LIN {X 0.158,Y -379.626,Z 827.651,A 0.000,B 0.000,C 90.000,E1 153.127} C_DIS
LIN {X -0.056,Y -381.140,Z 827.648,A 0.000,B 0.000,C 90.000,E1 152.615} C_DIS
LIN {X 0.104,Y -381.893,Z 827.647,A 0.000,B 0.000,C 90.000,E1 152.410} C_DIS
LIN {X 0.072,Y -384.199,Z 827.643,A 0.000,B 0.000,C 90.000,E1 151.691} C_DIS
LIN {X 0.062,Y -387.788,Z 827.639,A 0.000,B 0.000,C 90.000,E1 150.973} C_DIS
LIN {X 0.027,Y -391.705,Z 827.636,A 0.000,B 0.000,C 90.000,E1 150.383} C_DIS
LIN {X 0.218,Y -394.693,Z 827.634,A 0.000,B 0.000,C 90.000,E1 149.999} C_DIS
LIN {X 0.081,Y -399.557,Z 827.631,A 0.000,B 0.000,C 90.000,E1 149.537} C_DIS
LIN {X -0.054,Y -401.389,Z 827.630,A 0.000,B 0.000,C 90.000,E1 149.410} C_DIS
LIN {X -0.036,Y -407.802,Z 827.628,A 0.000,B 0.000,C 90.000,E1 148.997} C_DIS
LIN {X -0.157,Y -417.907,Z 827.625,A 0.000,B 0.000,C 90.000,E1 148.456} C_DIS
LIN {X -0.139,Y -427.004,Z 827.622,A 0.000,B 0.000,C 90.000,E1 147.995} C_DIS
LIN {X -0.155,Y -435.286,Z 827.620,A 0.000,B 0.000,C 90.000,E1 147.533} C_DIS
LIN {X -0.107,Y -441.668,Z 827.617,A 0.000,B 0.000,C 90.000,E1 147.120} C_DIS
LIN {X 0.193,Y -449.116,Z 827.614,A 0.000,B 0.000,C 90.000,E1 146.501} C_DIS
LIN {X 0.115,Y -453.669,Z 827.612,A 0.000,B 0.000,C 90.000,E1 146.135} C_DIS
LIN {X -0.065,Y -463.952,Z 827.607,A 0.000,B 0.000,C 90.000,E1 145.229} C_DIS
LIN {X -0.066,Y -468.086,Z 827.605,A 0.000,B 0.000,C 90.000,E1 144.815} C_DIS
LIN {X 0.151,Y -473.259,Z 827.601,A 0.000,B 0.000,C 90.000,E1 144.196} C_DIS
LIN {X -0.013,Y -481.998,Z 827.595,A 0.000,B 0.000,C 90.000,E1 143.130} C_DIS
LIN {X 0.058,Y -487.602,Z 827.591,A 0.000,B 0.000,C 90.000,E1 142.351} C_DIS
LIN {X -0.130,Y -494.117,Z 827.586,A 0.000,B 0.000,C 90.000,E1 141.457} C_DIS
LIN {X 0.236,Y -501.224,Z 827.580,A 0.000,B 0.000,C 90.000,E1 140.356} C_DIS
LIN {X 0.094,Y -508.483,Z 827.573,A 0.000,B 0.000,C 90.000,E1 139.175} C_DIS
LIN {X -0.252,Y -513.528,Z 827.568,A 0.000,B 0.000,C 90.000,E1 138.324} C_DIS
LIN {X 0.133,Y -515.933,Z 827.566,A 0.000,B 0.000,C 90.000,E1 137.838} C_DIS
LIN {X 0.247,Y -524.458,Z 827.557,A 0.000,B 0.000,C 90.000,E1 136.215} C_DIS
LIN {X 0.280,Y -528.245,Z 827.553,A 0.000,B 0.000,C 90.000,E1 135.486} C_DIS
LIN {X 0.277,Y -534.712,Z 827.546,A 0.000,B 0.000,C 90.000,E1 134.190} C_DIS
LIN {X 0.004,Y -539.742,Z 827.540,A 0.000,B 0.000,C 90.000,E1 133.218} C_DIS
LIN {X -0.371,Y -546.176,Z 827.532,A 0.000,B 0.000,C 90.000,E1 131.838} C_DIS
LIN {X 0.101,Y -549.719,Z 827.528,A 0.000,B 0.000,C 90.000,E1 130.943} C_DIS
LIN {X -0.174,Y -554.151,Z 827.521,A 0.000,B 0.000,C 90.000,E1 129.850} C_DIS
LIN {X 0.111,Y -558.207,Z 827.515,A 0.000,B 0.000,C 90.000,E1 128.705} C_DIS
LIN {X -0.068,Y -560.940,Z 827.510,A 0.000,B 0.000,C 90.000,E1 127.890} C_DIS
LIN {X -0.225,Y -563.574,Z 827.506,A 0.000,B 0.000,C 90.000,E1 127.076} C_DIS
LIN {X 0.093,Y -565.796,Z 827.501,A 0.000,B 0.000,C 90.000,E1 126.217} C_DIS
LIN {X -0.014,Y -567.045,Z 827.498,A 0.000,B 0.000,C 90.000,E1 125.678} C_DIS
LIN {X -0.327,Y -568.955,Z 827.492,A 0.000,B 0.000,C 90.000,E1 124.612} C_DIS
LIN {X -0.152,Y -570.425,Z 827.486,A 0.000,B 0.000,C 90.000,E1 123.499} C_DIS
LIN {X -0.144,Y -571.632,Z 827.479,A 0.000,B 0.000,C 90.000,E1 122.133} C_DIS
LIN {X -0.372,Y -571.977,Z 827.474,A 0.000,B 0.000,C 90.000,E1 121.337} C_DIS
LIN {X 0.192,Y -571.764,Z 827.469,A 0.000,B 0.000,C 90.000,E1 120.463} C_DIS
LIN {X 0.139,Y -571.928,Z 827.466,A 0.000,B 0.000,C 90.000,E1 119.922} C_DIS
LIN {X -0.198,Y -571.755,Z 827.463,A 0.000,B 0.000,C 90.000,E1 119.411} C_DIS
LIN {X 0.245,Y -571.352,Z 827.460,A 0.000,B 0.000,C 90.000,E1 118.821} C_DIS
LIN {X 0.182,Y -570.016,Z 827.453,A 0.000,B 0.000,C 90.000,E1 117.462} C_DIS
LIN {X 0.013,Y -569.716,Z 827.451,A 0.000,B 0.000,C 90.000,E1 117.206} C_DIS
LIN {X 0.264,Y -568.037,Z 827.447,A 0.000,B 0.000,C 90.000,E1 116.360} C_DIS
LIN {X -0.266,Y -566.017,Z 827.442,A 0.000,B 0.000,C 90.000,E1 115.591} C_DIS
LIN {X 0.063,Y -565.403,Z 827.441,A 0.000,B 0.000,C 90.000,E1 115.283} C_DIS
LIN {X -0.077,Y -562.630,Z 827.435,A 0.000,B 0.000,C 90.000,E1 114.335} C_DIS
LIN {X -0.174,Y -562.501,Z 827.434,A 0.000,B 0.000,C 90.000,E1 114.207} C_DIS
LIN {X 0.056,Y -562.518,Z 827.434,A 0.000,B 0.000,C 90.000,E1 114.027} C_DIS
LIN {X -0.142,Y -562.013,Z 827.432,A 0.000,B 0.000,C 90.000,E1 113.770} C_DIS
LIN {X 0.177,Y -562.133,Z 827.430,A 0.000,B 0.000,C 90.000,E1 113.462} C_DIS
LIN {X -0.023,Y -561.934,Z 827.429,A 0.000,B 0.000,C 90.000,E1 113.206} C_DIS
LIN {X -0.063,Y -561.520,Z 827.428,A 0.000,B 0.000,C 90.000,E1 113.003} C_DIS
LIN {X 0.091,Y -561.775,Z 827.426,A 0.000,B 0.000,C 90.000,E1 112.642} C_DIS
LIN {X -0.213,Y -561.989,Z 827.421,A 0.000,B 0.000,C 90.000,E1 111.844} C_DIS
LIN {X 0.214,Y -562.412,Z 827.417,A 0.000,B 0.000,C 90.000,E1 110.972} C_DIS
LIN {X -0.173,Y -562.591,Z 827.409,A 0.000,B 0.000,C 90.000,E1 109.631} C_DIS
LIN {X -0.201,Y -562.482,Z 827.395,A 0.000,B 0.000,C 90.000,E1 107.149} C_DIS
LIN {X -0.108,Y -563.355,Z 827.377,A 0.000,B 0.000,C 90.000,E1 103.828} C_DIS
LIN {X -0.124,Y -564.958,Z 827.362,A 0.000,B 0.000,C 90.000,E1 101.074} C_DIS
LIN {X -0.229,Y -566.219,Z 827.352,A 0.000,B 0.000,C 90.000,E1 99.434} C_DIS
LIN {X 0.057,Y -567.336,Z 827.343,A 0.000,B 0.000,C 90.000,E1 97.757} C_DIS
LIN {X -0.261,Y -568.305,Z 827.334,A 0.000,B 0.000,C 90.000,E1 96.144} C_DIS
LIN {X -0.106,Y -568.991,Z 827.326,A 0.000,B 0.000,C 90.000,E1 94.759} C_DIS
LIN {X -0.036,Y -569.598,Z 827.319,A 0.000,B 0.000,C 90.000,E1 93.383} C_DIS
LIN {X 0.057,Y -570.037,Z 827.311,A 0.000,B 0.000,C 90.000,E1 92.007} C_DIS
LIN {X 0.154,Y -570.510,Z 827.304,A 0.000,B 0.000,C 90.000,E1 90.630} C_DIS
LIN {X -0.193,Y -570.931,Z 827.295,A 0.000,B 0.000,C 90.000,E1 89.026} C_DIS
LIN {X -0.082,Y -571.308,Z 827.287,A 0.000,B 0.000,C 90.000,E1 87.650} C_DIS
LIN {X -0.236,Y -571.670,Z 827.276,A 0.000,B 0.000,C 90.000,E1 85.755} C_DIS
LIN {X -0.073,Y -571.889,Z 827.269,A 0.000,B 0.000,C 90.000,E1 84.375} C_DIS
LIN {X 0.271,Y -572.275,Z 827.260,A 0.000,B 0.000,C 90.000,E1 82.704} C_DIS
LIN {X -0.052,Y -572.772,Z 827.248,A 0.000,B 0.000,C 90.000,E1 80.557} C_DIS
LIN {X 0.274,Y -573.188,Z 827.240,A 0.000,B 0.000,C 90.000,E1 79.162} C_DIS
LIN {X 0.031,Y -573.590,Z 827.232,A 0.000,B 0.000,C 90.000,E1 77.825} C_DIS
LIN {X 0.038,Y -573.823,Z 827.225,A 0.000,B 0.000,C 90.000,E1 76.464} C_DIS
LIN {X 0.257,Y -574.035,Z 827.216,A 0.000,B 0.000,C 90.000,E1 74.810} C_DIS
LIN {X -0.278,Y -574.043,Z 827.208,A 0.000,B 0.000,C 90.000,E1 73.504} C_DIS
LIN {X -0.103,Y -574.028,Z 827.201,A 0.000,B 0.000,C 90.000,E1 72.127} C_DIS
LIN {X 0.249,Y -573.869,Z 827.193,A 0.000,B 0.000,C 90.000,E1 70.732} C_DIS
LIN {X 0.047,Y -573.554,Z 827.183,A 0.000,B 0.000,C 90.000,E1 68.847} C_DIS
LIN {X -0.112,Y -573.131,Z 827.173,A 0.000,B 0.000,C 90.000,E1 67.230} C_DIS
LIN {X -0.112,Y -572.685,Z 827.166,A 0.000,B 0.000,C 90.000,E1 65.869} C_DIS
LIN {X -0.250,Y -572.259,Z 827.160,A 0.000,B 0.000,C 90.000,E1 64.793} C_DIS
LIN {X 0.044,Y -571.456,Z 827.151,A 0.000,B 0.000,C 90.000,E1 63.127} C_DIS
LIN {X -0.018,Y -570.640,Z 827.143,A 0.000,B 0.000,C 90.000,E1 61.769} C_DIS
LIN {X 0.073,Y -569.770,Z 827.137,A 0.000,B 0.000,C 90.000,E1 60.667} C_DIS
LIN {X -0.171,Y -568.952,Z 827.133,A 0.000,B 0.000,C 90.000,E1 59.871} C_DIS
LIN {X 0.173,Y -567.724,Z 827.126,A 0.000,B 0.000,C 90.000,E1 58.742} C_DIS
LIN {X 0.014,Y -566.317,Z 827.120,A 0.000,B 0.000,C 90.000,E1 57.661} C_DIS
LIN {X 0.144,Y -564.684,Z 827.114,A 0.000,B 0.000,C 90.000,E1 56.548} C_DIS
LIN {X 0.152,Y -563.325,Z 827.110,A 0.000,B 0.000,C 90.000,E1 55.722} C_DIS
LIN {X 0.143,Y -561.776,Z 827.105,A 0.000,B 0.000,C 90.000,E1 54.895} C_DIS
LIN {X 0.206,Y -559.363,Z 827.099,A 0.000,B 0.000,C 90.000,E1 53.783} C_DIS
LIN {X 0.030,Y -557.395,Z 827.094,A 0.000,B 0.000,C 90.000,E1 52.970} C_DIS
LIN {X 0.200,Y -555.953,Z 827.091,A 0.000,B 0.000,C 90.000,E1 52.396} C_DIS
LIN {X -0.002,Y -553.554,Z 827.087,A 0.000,B 0.000,C 90.000,E1 51.582} C_DIS
LIN {X 0.203,Y -550.838,Z 827.082,A 0.000,B 0.000,C 90.000,E1 50.723} C_DIS
LIN {X -0.053,Y -547.802,Z 827.077,A 0.000,B 0.000,C 90.000,E1 49.908} C_DIS
LIN {X 0.035,Y -545.676,Z 827.074,A 0.000,B 0.000,C 90.000,E1 49.337} C_DIS
LIN {X 0.077,Y -541.954,Z 827.069,A 0.000,B 0.000,C 90.000,E1 48.485} C_DIS
LIN {X 0.066,Y -539.294,Z 827.066,A 0.000,B 0.000,C 90.000,E1 47.919} C_DIS
LIN {X -0.320,Y -536.391,Z 827.063,A 0.000,B 0.000,C 90.000,E1 47.391} C_DIS
LIN {X 0.198,Y -532.300,Z 827.059,A 0.000,B 0.000,C 90.000,E1 46.620} C_DIS
LIN {X 0.126,Y -528.699,Z 827.056,A 0.000,B 0.000,C 90.000,E1 46.053} C_DIS
LIN {X 0.029,Y -524.808,Z 827.053,A 0.000,B 0.000,C 90.000,E1 45.486} C_DIS
LIN {X -0.089,Y -520.511,Z 827.050,A 0.000,B 0.000,C 90.000,E1 44.919} C_DIS
LIN {X -0.014,Y -517.102,Z 827.047,A 0.000,B 0.000,C 90.000,E1 44.474} C_DIS
LIN {X 0.175,Y -512.157,Z 827.044,A 0.000,B 0.000,C 90.000,E1 43.866} C_DIS
LIN {X 0.016,Y -506.901,Z 827.041,A 0.000,B 0.000,C 90.000,E1 43.299} C_DIS
LIN {X 0.165,Y -502.891,Z 827.038,A 0.000,B 0.000,C 90.000,E1 42.852} C_DIS
LIN {X -0.018,Y -494.404,Z 827.034,A 0.000,B 0.000,C 90.000,E1 42.043} C_DIS
LIN {X -0.116,Y -486.930,Z 827.030,A 0.000,B 0.000,C 90.000,E1 41.391} C_DIS
LIN {X 0.099,Y -477.756,Z 827.026,A 0.000,B 0.000,C 90.000,E1 40.620} C_DIS
LIN {X 0.063,Y -469.888,Z 827.022,A 0.000,B 0.000,C 90.000,E1 40.011} C_DIS
LIN {X 0.018,Y -458.832,Z 827.018,A 0.000,B 0.000,C 90.000,E1 39.197} C_DIS
LIN {X 0.144,Y -442.903,Z 827.011,A 0.000,B 0.000,C 90.000,E1 38.016} C_DIS
LIN {X -0.087,Y -419.409,Z 827.001,A 0.000,B 0.000,C 90.000,E1 36.217} C_DIS
LIN {X -0.110,Y -405.927,Z 826.995,A 0.000,B 0.000,C 90.000,E1 35.025} C_DIS
LIN {X -0.100,Y -400.639,Z 826.992,A 0.000,B 0.000,C 90.000,E1 34.485} C_DIS
LIN {X 0.175,Y -397.087,Z 826.989,A 0.000,B 0.000,C 90.000,E1 33.992} C_DIS
LIN {X 0.136,Y -397.070,Z 826.989,A 0.000,B 0.000,C 90.000,E1 33.992} C_DIS
LIN {X 0.141,Y -393.525,Z 826.976,A 0.000,B 0.000,C 90.000,E1 31.671} C_DIS
LIN {X 0.136,Y -391.963,Z 826.972,A 0.000,B 0.000,C 90.000,E1 30.875} C_DIS
LIN {X 0.067,Y -391.882,Z 826.971,A 0.000,B 0.000,C 90.000,E1 30.797} C_DIS
LIN {X 0.021,Y -393.684,Z 826.951,A 0.000,B 0.000,C 90.000,E1 27.078} C_DIS
LIN {X -0.061,Y -395.561,Z 826.935,A 0.000,B 0.000,C 90.000,E1 24.259} C_DIS
LIN {X -0.131,Y -397.199,Z 826.923,A 0.000,B 0.000,C 90.000,E1 22.153} C_DIS
LIN {X -0.014,Y -399.623,Z 826.907,A 0.000,B 0.000,C 90.000,E1 19.322} C_DIS
LIN {X 0.166,Y -402.678,Z 826.892,A 0.000,B 0.000,C 90.000,E1 16.496} C_DIS
LIN {X -0.165,Y -407.528,Z 826.872,A 0.000,B 0.000,C 90.000,E1 13.063} C_DIS
LIN {X 0.173,Y -412.017,Z 826.857,A 0.000,B 0.000,C 90.000,E1 10.254} C_DIS
LIN {X -0.001,Y -415.629,Z 826.846,A 0.000,B 0.000,C 90.000,E1 8.219} C_DIS
LIN {X 0.199,Y -418.690,Z 826.836,A 0.000,B 0.000,C 90.000,E1 6.486} C_DIS
LIN {X 0.057,Y -423.009,Z 826.823,A 0.000,B 0.000,C 90.000,E1 4.131} C_DIS
LIN {X 0.036,Y -427.709,Z 826.810,A 0.000,B 0.000,C 90.000,E1 1.776} C_DIS
LIN {X -0.020,Y -434.217,Z 826.793,A 0.000,B 0.000,C 90.000,E1 358.797} C_DIS
LIN {X 0.151,Y -438.864,Z 826.782,A 0.000,B 0.000,C 90.000,E1 356.788} C_DIS
LIN {X -0.116,Y -442.925,Z 826.773,A 0.000,B 0.000,C 90.000,E1 355.179} C_DIS
LIN {X -0.142,Y -447.878,Z 826.762,A 0.000,B 0.000,C 90.000,E1 353.223} C_DIS
LIN {X -0.146,Y -452.367,Z 826.753,A 0.000,B 0.000,C 90.000,E1 351.602} C_DIS
LIN {X 0.126,Y -454.113,Z 826.751,A 0.000,B 0.000,C 90.000,E1 351.084} C_DIS
LIN {X -0.113,Y -455.583,Z 826.749,A 0.000,B 0.000,C 90.000,E1 350.792} C_DIS
LIN {X -0.042,Y -456.513,Z 826.748,A 0.000,B 0.000,C 90.000,E1 350.622} C_DIS
LIN {X 0.095,Y -458.920,Z 826.746,A 0.000,B 0.000,C 90.000,E1 350.274} C_DIS
LIN {X -0.144,Y -461.863,Z 826.744,A 0.000,B 0.000,C 90.000,E1 349.982} C_DIS
LIN {X 0.139,Y -467.280,Z 826.742,A 0.000,B 0.000,C 90.000,E1 349.511} C_DIS
LIN {X -0.155,Y -475.770,Z 826.739,A 0.000,B 0.000,C 90.000,E1 348.993} C_DIS
LIN {X -0.103,Y -488.891,Z 826.734,A 0.000,B 0.000,C 90.000,E1 348.173} C_DIS
LIN {X 0.094,Y -504.918,Z 826.729,A 0.000,B 0.000,C 90.000,E1 347.117} C_DIS
LIN {X -0.200,Y -514.264,Z 826.725,A 0.000,B 0.000,C 90.000,E1 346.520} C_DIS
LIN {X -0.122,Y -526.667,Z 826.720,A 0.000,B 0.000,C 90.000,E1 345.644} C_DIS
LIN {X -0.231,Y -535.675,Z 826.717,A 0.000,B 0.000,C 90.000,E1 344.991} C_DIS
LIN {X -0.012,Y -544.484,Z 826.713,A 0.000,B 0.000,C 90.000,E1 344.283} C_DIS
LIN {X 0.043,Y -551.586,Z 826.709,A 0.000,B 0.000,C 90.000,E1 343.685} C_DIS
LIN {X -0.135,Y -558.409,Z 826.706,A 0.000,B 0.000,C 90.000,E1 343.087} C_DIS
LIN {X 0.238,Y -563.727,Z 826.703,A 0.000,B 0.000,C 90.000,E1 342.543} C_DIS
LIN {X -0.314,Y -570.002,Z 826.700,A 0.000,B 0.000,C 90.000,E1 341.945} C_DIS
LIN {X -0.233,Y -574.905,Z 826.697,A 0.000,B 0.000,C 90.000,E1 341.402} C_DIS
LIN {X 0.043,Y -578.475,Z 826.694,A 0.000,B 0.000,C 90.000,E1 340.967} C_DIS
LIN {X -0.278,Y -584.902,Z 826.690,A 0.000,B 0.000,C 90.000,E1 340.188} C_DIS
LIN {X -0.276,Y -589.853,Z 826.686,A 0.000,B 0.000,C 90.000,E1 339.518} C_DIS
LIN {X -0.018,Y -594.338,Z 826.682,A 0.000,B 0.000,C 90.000,E1 338.827} C_DIS
LIN {X -0.244,Y -600.170,Z 826.677,A 0.000,B 0.000,C 90.000,E1 337.922} C_DIS
LIN {X 0.050,Y -605.603,Z 826.672,A 0.000,B 0.000,C 90.000,E1 336.975} C_DIS
LIN {X 0.157,Y -611.642,Z 826.666,A 0.000,B 0.000,C 90.000,E1 335.921} C_DIS
LIN {X -0.212,Y -616.711,Z 826.661,A 0.000,B 0.000,C 90.000,E1 335.049} C_DIS
LIN {X -0.268,Y -622.133,Z 826.656,A 0.000,B 0.000,C 90.000,E1 334.024} C_DIS
LIN {X -0.258,Y -625.952,Z 826.651,A 0.000,B 0.000,C 90.000,E1 333.256} C_DIS
LIN {X -0.212,Y -629.576,Z 826.647,A 0.000,B 0.000,C 90.000,E1 332.487} C_DIS
LIN {X 0.235,Y -635.207,Z 826.640,A 0.000,B 0.000,C 90.000,E1 331.179} C_DIS
LIN {X -0.192,Y -638.553,Z 826.636,A 0.000,B 0.000,C 90.000,E1 330.461} C_DIS
LIN {X -0.210,Y -642.760,Z 826.630,A 0.000,B 0.000,C 90.000,E1 329.459} C_DIS
LIN {X 0.313,Y -645.746,Z 826.626,A 0.000,B 0.000,C 90.000,E1 328.663} C_DIS
LIN {X -0.157,Y -649.350,Z 826.621,A 0.000,B 0.000,C 90.000,E1 327.709} C_DIS
LIN {X -0.037,Y -652.768,Z 826.615,A 0.000,B 0.000,C 90.000,E1 326.707} C_DIS
LIN {X 0.029,Y -656.724,Z 826.608,A 0.000,B 0.000,C 90.000,E1 325.468} C_DIS
LIN {X 0.040,Y -658.162,Z 826.605,A 0.000,B 0.000,C 90.000,E1 324.975} C_DIS
LIN {X 0.092,Y -660.874,Z 826.600,A 0.000,B 0.000,C 90.000,E1 323.989} C_DIS
LIN {X 0.176,Y -663.377,Z 826.595,A 0.000,B 0.000,C 90.000,E1 323.004} C_DIS
LIN {X -0.267,Y -666.235,Z 826.588,A 0.000,B 0.000,C 90.000,E1 321.823} C_DIS
LIN {X -0.216,Y -667.749,Z 826.584,A 0.000,B 0.000,C 90.000,E1 321.090} C_DIS
LIN {X -0.073,Y -670.596,Z 826.576,A 0.000,B 0.000,C 90.000,E1 319.622} C_DIS
LIN {X 0.031,Y -672.703,Z 826.569,A 0.000,B 0.000,C 90.000,E1 318.405} C_DIS
LIN {X -0.351,Y -674.357,Z 826.564,A 0.000,B 0.000,C 90.000,E1 317.472} C_DIS
LIN {X 0.215,Y -675.447,Z 826.560,A 0.000,B 0.000,C 90.000,E1 316.701} C_DIS
LIN {X 0.366,Y -677.090,Z 826.553,A 0.000,B 0.000,C 90.000,E1 315.486} C_DIS
LIN {X -0.008,Y -678.029,Z 826.549,A 0.000,B 0.000,C 90.000,E1 314.798} C_DIS
LIN {X -0.213,Y -679.943,Z 826.540,A 0.000,B 0.000,C 90.000,E1 313.137} C_DIS
LIN {X 0.084,Y -681.575,Z 826.532,A 0.000,B 0.000,C 90.000,E1 311.676} C_DIS
LIN {X 0.368,Y -682.868,Z 826.525,A 0.000,B 0.000,C 90.000,E1 310.458} C_DIS
LIN {X -0.337,Y -683.813,Z 826.520,A 0.000,B 0.000,C 90.000,E1 309.564} C_DIS
LIN {X 0.118,Y -685.070,Z 826.512,A 0.000,B 0.000,C 90.000,E1 308.096} C_DIS
LIN {X -0.194,Y -686.524,Z 826.503,A 0.000,B 0.000,C 90.000,E1 306.457} C_DIS
LIN {X 0.264,Y -687.475,Z 826.496,A 0.000,B 0.000,C 90.000,E1 305.231} C_DIS
LIN {X -0.055,Y -688.329,Z 826.489,A 0.000,B 0.000,C 90.000,E1 304.072} C_DIS
LIN {X 0.093,Y -689.695,Z 826.479,A 0.000,B 0.000,C 90.000,E1 302.163} C_DIS
LIN {X 0.045,Y -690.732,Z 826.471,A 0.000,B 0.000,C 90.000,E1 300.747} C_DIS
LIN {X 0.001,Y -691.745,Z 826.463,A 0.000,B 0.000,C 90.000,E1 299.333} C_DIS
LIN {X 0.230,Y -692.758,Z 826.455,A 0.000,B 0.000,C 90.000,E1 297.897} C_DIS
LIN {X -0.216,Y -694.091,Z 826.446,A 0.000,B 0.000,C 90.000,E1 296.283} C_DIS
LIN {X 0.106,Y -695.069,Z 826.439,A 0.000,B 0.000,C 90.000,E1 295.079} C_DIS
LIN {X -0.062,Y -695.667,Z 826.435,A 0.000,B 0.000,C 90.000,E1 294.387} C_DIS
LIN {X -0.224,Y -695.703,Z 826.432,A 0.000,B 0.000,C 90.000,E1 293.695} C_DIS
LIN {X 0.001,Y -694.815,Z 826.429,A 0.000,B 0.000,C 90.000,E1 293.206} C_DIS
LIN {X 0.249,Y -694.146,Z 826.428,A 0.000,B 0.000,C 90.000,E1 292.950} C_DIS
LIN {X 0.226,Y -692.688,Z 826.426,A 0.000,B 0.000,C 90.000,E1 292.717} C_DIS
LIN {X -0.055,Y -689.883,Z 826.424,A 0.000,B 0.000,C 90.000,E1 292.386} C_DIS
LIN {X -0.201,Y -688.713,Z 826.424,A 0.000,B 0.000,C 90.000,E1 292.280} C_DIS
LIN {X -0.087,Y -686.910,Z 826.423,A 0.000,B 0.000,C 90.000,E1 292.153} C_DIS
LIN {X 0.187,Y -681.422,Z 826.422,A 0.000,B 0.000,C 90.000,E1 291.844} C_DIS
LIN {X 0.130,Y -679.603,Z 826.421,A 0.000,B 0.000,C 90.000,E1 291.770} C_DIS
LIN {X 0.095,Y -671.476,Z 826.420,A 0.000,B 0.000,C 90.000,E1 291.535} C_DIS
LIN {X -0.183,Y -663.435,Z 826.419,A 0.000,B 0.000,C 90.000,E1 291.408} C_DIS
LIN {X 0.147,Y -650.714,Z 826.418,A 0.000,B 0.000,C 90.000,E1 291.173} C_DIS
LIN {X 0.197,Y -640.689,Z 826.417,A 0.000,B 0.000,C 90.000,E1 290.972} C_DIS
LIN {X -0.266,Y -631.460,Z 826.415,A 0.000,B 0.000,C 90.000,E1 290.791} C_DIS
LIN {X 0.177,Y -628.223,Z 826.415,A 0.000,B 0.000,C 90.000,E1 290.663} C_DIS
LIN {X -0.027,Y -621.652,Z 826.414,A 0.000,B 0.000,C 90.000,E1 290.429} C_DIS
LIN {X 0.046,Y -616.872,Z 826.412,A 0.000,B 0.000,C 90.000,E1 290.174} C_DIS
LIN {X -0.012,Y -616.790,Z 826.412,A 0.000,B 0.000,C 90.000,E1 290.174} C_DIS
LIN {X -0.125,Y -616.369,Z 826.412,A 0.000,B 0.000,C 90.000,E1 290.120} C_DIS
LIN {X 0.132,Y -614.944,Z 826.411,A 0.000,B 0.000,C 90.000,E1 289.939} C_DIS
LIN {X 0.090,Y -614.916,Z 826.411,A 0.000,B 0.000,C 90.000,E1 289.939} C_DIS
LIN {X 0.167,Y -614.913,Z 826.409,A 0.000,B 0.000,C 90.000,E1 289.577} C_DIS
LIN {X -0.064,Y -616.462,Z 826.407,A 0.000,B 0.000,C 90.000,E1 289.214} C_DIS
LIN {X -0.129,Y -618.606,Z 826.405,A 0.000,B 0.000,C 90.000,E1 288.833} C_DIS
LIN {X -0.044,Y -623.231,Z 826.400,A 0.000,B 0.000,C 90.000,E1 288.055} C_DIS
LIN {X 0.303,Y -625.859,Z 826.397,A 0.000,B 0.000,C 90.000,E1 287.511} C_DIS
LIN {X -0.129,Y -628.741,Z 826.394,A 0.000,B 0.000,C 90.000,E1 286.913} C_DIS
LIN {X 0.074,Y -630.848,Z 826.391,A 0.000,B 0.000,C 90.000,E1 286.386} C_DIS
LIN {X 0.285,Y -633.426,Z 826.387,A 0.000,B 0.000,C 90.000,E1 285.607} C_DIS
LIN {X -0.082,Y -634.876,Z 826.384,A 0.000,B 0.000,C 90.000,E1 285.134} C_DIS
LIN {X 0.164,Y -636.699,Z 826.380,A 0.000,B 0.000,C 90.000,E1 284.356} C_DIS
LIN {X -0.183,Y -637.506,Z 826.377,A 0.000,B 0.000,C 90.000,E1 283.883} C_DIS
LIN {X 0.098,Y -638.090,Z 826.374,A 0.000,B 0.000,C 90.000,E1 283.355} C_DIS
LIN {X 0.215,Y -638.578,Z 826.370,A 0.000,B 0.000,C 90.000,E1 282.591} C_DIS
LIN {X -0.120,Y -638.377,Z 826.367,A 0.000,B 0.000,C 90.000,E1 282.119} C_DIS
LIN {X -0.130,Y -637.692,Z 826.363,A 0.000,B 0.000,C 90.000,E1 281.366} C_DIS
LIN {X 0.156,Y -636.847,Z 826.360,A 0.000,B 0.000,C 90.000,E1 280.838} C_DIS
LIN {X -0.194,Y -635.687,Z 826.358,A 0.000,B 0.000,C 90.000,E1 280.366} C_DIS
LIN {X -0.040,Y -634.119,Z 826.355,A 0.000,B 0.000,C 90.000,E1 279.849} C_DIS
LIN {X 0.214,Y -632.324,Z 826.352,A 0.000,B 0.000,C 90.000,E1 279.321} C_DIS
LIN {X -0.078,Y -631.298,Z 826.351,A 0.000,B 0.000,C 90.000,E1 279.095} C_DIS
LIN {X 0.149,Y -628.733,Z 826.348,A 0.000,B 0.000,C 90.000,E1 278.568} C_DIS
LIN {X 0.262,Y -625.774,Z 826.345,A 0.000,B 0.000,C 90.000,E1 278.049} C_DIS
LIN {X -0.261,Y -622.418,Z 826.342,A 0.000,B 0.000,C 90.000,E1 277.587} C_DIS
LIN {X 0.127,Y -620.282,Z 826.341,A 0.000,B 0.000,C 90.000,E1 277.296} C_DIS
LIN {X -0.269,Y -616.889,Z 826.339,A 0.000,B 0.000,C 90.000,E1 276.947} C_DIS
LIN {X -0.035,Y -612.955,Z 826.336,A 0.000,B 0.000,C 90.000,E1 276.549} C_DIS
LIN {X -0.025,Y -611.631,Z 826.336,A 0.000,B 0.000,C 90.000,E1 276.429} C_DIS
LIN {X -0.016,Y -607.028,Z 826.334,A 0.000,B 0.000,C 90.000,E1 276.087} C_DIS
LIN {X -0.173,Y -601.929,Z 826.332,A 0.000,B 0.000,C 90.000,E1 275.796} C_DIS
LIN {X 0.259,Y -593.679,Z 826.330,A 0.000,B 0.000,C 90.000,E1 275.334} C_DIS
LIN {X -0.274,Y -589.760,Z 826.329,A 0.000,B 0.000,C 90.000,E1 275.220} C_DIS
LIN {X -0.163,Y -582.790,Z 826.327,A 0.000,B 0.000,C 90.000,E1 274.935} C_DIS
LIN {X 0.303,Y -579.263,Z 826.327,A 0.000,B 0.000,C 90.000,E1 274.759} C_DIS
LIN {X 0.203,Y -574.617,Z 826.326,A 0.000,B 0.000,C 90.000,E1 274.645} C_DIS
LIN {X -0.257,Y -572.579,Z 826.326,A 0.000,B 0.000,C 90.000,E1 274.645} C_DIS
LIN {X -0.018,Y -566.191,Z 826.325,A 0.000,B 0.000,C 90.000,E1 274.531} C_DIS
LIN {X -0.161,Y -560.220,Z 826.325,A 0.000,B 0.000,C 90.000,E1 274.531} C_DIS
LIN {X -0.215,Y -552.833,Z 826.325,A 0.000,B 0.000,C 90.000,E1 274.531} C_DIS
LIN {X -0.011,Y -550.583,Z 826.325,A 0.000,B 0.000,C 90.000,E1 274.473} C_DIS
LIN {X -0.047,Y -550.467,Z 826.325,A 0.000,B 0.000,C 90.000,E1 274.473} C_DIS
LIN {X 0.196,Y -549.604,Z 826.323,A 0.000,B 0.000,C 90.000,E1 274.131} C_DIS
LIN {X -0.083,Y -548.612,Z 826.318,A 0.000,B 0.000,C 90.000,E1 273.326} C_DIS
LIN {X 0.185,Y -547.475,Z 826.311,A 0.000,B 0.000,C 90.000,E1 271.892} C_DIS
LIN {X -0.077,Y -546.245,Z 826.301,A 0.000,B 0.000,C 90.000,E1 270.229} C_DIS
LIN {X 0.168,Y -545.050,Z 826.292,A 0.000,B 0.000,C 90.000,E1 268.511} C_DIS
LIN {X -0.064,Y -543.522,Z 826.279,A 0.000,B 0.000,C 90.000,E1 266.274} C_DIS
LIN {X 0.137,Y -542.611,Z 826.271,A 0.000,B 0.000,C 90.000,E1 264.837} C_DIS
LIN {X -0.234,Y -541.851,Z 826.265,A 0.000,B 0.000,C 90.000,E1 263.742} C_DIS
LIN {X -0.080,Y -540.921,Z 826.259,A 0.000,B 0.000,C 90.000,E1 262.591} C_DIS
LIN {X 0.268,Y -539.328,Z 826.249,A 0.000,B 0.000,C 90.000,E1 260.849} C_DIS
LIN {X -0.010,Y -537.954,Z 826.241,A 0.000,B 0.000,C 90.000,E1 259.454} C_DIS
LIN {X -0.150,Y -536.222,Z 826.232,A 0.000,B 0.000,C 90.000,E1 257.757} C_DIS
LIN {X 0.079,Y -535.140,Z 826.226,A 0.000,B 0.000,C 90.000,E1 256.589} C_DIS
LIN {X 0.163,Y -532.853,Z 826.214,A 0.000,B 0.000,C 90.000,E1 254.574} C_DIS
LIN {X 0.152,Y -530.882,Z 826.205,A 0.000,B 0.000,C 90.000,E1 252.851} C_DIS
LIN {X 0.050,Y -529.471,Z 826.198,A 0.000,B 0.000,C 90.000,E1 251.710} C_DIS
LIN {X 0.276,Y -527.625,Z 826.190,A 0.000,B 0.000,C 90.000,E1 250.242} C_DIS
LIN {X -0.013,Y -525.635,Z 826.182,A 0.000,B 0.000,C 90.000,E1 248.827} C_DIS
LIN {X -0.010,Y -522.753,Z 826.171,A 0.000,B 0.000,C 90.000,E1 246.794} C_DIS
LIN {X -0.190,Y -520.477,Z 826.163,A 0.000,B 0.000,C 90.000,E1 245.357} C_DIS
LIN {X -0.062,Y -517.616,Z 826.153,A 0.000,B 0.000,C 90.000,E1 243.589} C_DIS
LIN {X 0.106,Y -515.067,Z 826.145,A 0.000,B 0.000,C 90.000,E1 242.103} C_DIS
LIN {X 0.124,Y -512.926,Z 826.139,A 0.000,B 0.000,C 90.000,E1 240.923} C_DIS
LIN {X 0.088,Y -509.727,Z 826.129,A 0.000,B 0.000,C 90.000,E1 239.154} C_DIS
LIN {X -0.151,Y -507.450,Z 826.122,A 0.000,B 0.000,C 90.000,E1 237.995} C_DIS
LIN {X -0.034,Y -505.655,Z 826.117,A 0.000,B 0.000,C 90.000,E1 237.089} C_DIS
LIN {X -0.130,Y -501.766,Z 826.107,A 0.000,B 0.000,C 90.000,E1 235.308} C_DIS
LIN {X -0.041,Y -497.615,Z 826.097,A 0.000,B 0.000,C 90.000,E1 233.497} C_DIS
LIN {X -0.160,Y -493.287,Z 826.087,A 0.000,B 0.000,C 90.000,E1 231.698} C_DIS
LIN {X 0.242,Y -490.364,Z 826.080,A 0.000,B 0.000,C 90.000,E1 230.436} C_DIS
LIN {X 0.028,Y -485.381,Z 826.069,A 0.000,B 0.000,C 90.000,E1 228.324} C_DIS
LIN {X 0.200,Y -481.161,Z 826.058,A 0.000,B 0.000,C 90.000,E1 226.458} C_DIS
LIN {X 0.034,Y -476.526,Z 826.046,A 0.000,B 0.000,C 90.000,E1 224.312} C_DIS
LIN {X -0.136,Y -471.161,Z 826.032,A 0.000,B 0.000,C 90.000,E1 221.838} C_DIS
LIN {X 0.247,Y -465.855,Z 826.018,A 0.000,B 0.000,C 90.000,E1 219.277} C_DIS
LIN {X 0.224,Y -463.209,Z 826.011,A 0.000,B 0.000,C 90.000,E1 218.016} C_DIS
LIN {X 0.004,Y -459.260,Z 826.001,A 0.000,B 0.000,C 90.000,E1 216.137} C_DIS
LIN {X 0.065,Y -455.969,Z 825.992,A 0.000,B 0.000,C 90.000,E1 214.532} C_DIS
LIN {X 0.090,Y -450.527,Z 825.978,A 0.000,B 0.000,C 90.000,E1 211.957} C_DIS
LIN {X 0.191,Y -446.507,Z 825.967,A 0.000,B 0.000,C 90.000,E1 210.001} C_DIS
LIN {X -0.251,Y -442.665,Z 825.956,A 0.000,B 0.000,C 90.000,E1 208.103} C_DIS
LIN {X -0.036,Y -439.411,Z 825.947,A 0.000,B 0.000,C 90.000,E1 206.437} C_DIS
LIN {X 0.094,Y -436.824,Z 825.940,A 0.000,B 0.000,C 90.000,E1 205.103} C_DIS
LIN {X 0.001,Y -432.766,Z 825.929,A 0.000,B 0.000,C 90.000,E1 203.131} C_DIS
LIN {X 0.068,Y -428.259,Z 825.916,A 0.000,B 0.000,C 90.000,E1 200.791} C_DIS
LIN {X 0.079,Y -425.706,Z 825.908,A 0.000,B 0.000,C 90.000,E1 199.450} C_DIS
LIN {X -0.119,Y -421.709,Z 825.897,A 0.000,B 0.000,C 90.000,E1 197.457} C_DIS
LIN {X 0.055,Y -419.086,Z 825.889,A 0.000,B 0.000,C 90.000,E1 196.079} C_DIS
LIN {X -0.134,Y -415.269,Z 825.878,A 0.000,B 0.000,C 90.000,E1 194.064} C_DIS
LIN {X -0.144,Y -411.980,Z 825.869,A 0.000,B 0.000,C 90.000,E1 192.355} C_DIS
LIN {X 0.115,Y -407.996,Z 825.857,A 0.000,B 0.000,C 90.000,E1 190.254} C_DIS
LIN {X 0.197,Y -404.737,Z 825.847,A 0.000,B 0.000,C 90.000,E1 188.511} C_DIS
LIN {X 0.089,Y -400.221,Z 825.834,A 0.000,B 0.000,C 90.000,E1 186.087} C_DIS
LIN {X -0.105,Y -393.263,Z 825.810,A 0.000,B 0.000,C 90.000,E1 181.892} C_DIS
LIN {X -0.020,Y -389.051,Z 825.793,A 0.000,B 0.000,C 90.000,E1 178.682} C_DIS
LIN {X 0.015,Y -387.304,Z 825.785,A 0.000,B 0.000,C 90.000,E1 177.249} C_DIS
LIN {X 0.129,Y -384.310,Z 825.771,A 0.000,B 0.000,C 90.000,E1 174.723} C_DIS
LIN {X -0.038,Y -380.329,Z 825.751,A 0.000,B 0.000,C 90.000,E1 171.141} C_DIS
LIN {X 0.021,Y -377.651,Z 825.735,A 0.000,B 0.000,C 90.000,E1 168.229} C_DIS
LIN {X 0.105,Y -374.906,Z 825.716,A 0.000,B 0.000,C 90.000,E1 164.936} C_DIS
LIN {X 0.014,Y -372.888,Z 825.690,A 0.000,B 0.000,C 90.000,E1 160.188} C_DIS
LIN {X 0.123,Y -373.074,Z 825.680,A 0.000,B 0.000,C 90.000,E1 158.337} C_DIS
LIN {X 0.129,Y -373.666,Z 825.672,A 0.000,B 0.000,C 90.000,E1 156.869} C_DIS
LIN {X -0.023,Y -374.549,Z 825.666,A 0.000,B 0.000,C 90.000,E1 155.793} C_DIS
LIN {X 0.058,Y -375.424,Z 825.661,A 0.000,B 0.000,C 90.000,E1 155.049} C_DIS
LIN {X -0.071,Y -377.105,Z 825.655,A 0.000,B 0.000,C 90.000,E1 153.973} C_DIS
LIN {X 0.057,Y -377.851,Z 825.653,A 0.000,B 0.000,C 90.000,E1 153.589} C_DIS
LIN {X -0.149,Y -378.437,Z 825.651,A 0.000,B 0.000,C 90.000,E1 153.256} C_DIS
LIN {X 0.126,Y -380.216,Z 825.647,A 0.000,B 0.000,C 90.000,E1 152.487} C_DIS
LIN {X 0.082,Y -382.267,Z 825.643,A 0.000,B 0.000,C 90.000,E1 151.769} C_DIS
LIN {X -0.118,Y -384.287,Z 825.640,A 0.000,B 0.000,C 90.000,E1 151.257} C_DIS
LIN {X -0.120,Y -386.812,Z 825.637,A 0.000,B 0.000,C 90.000,E1 150.717} C_DIS
LIN {X -0.111,Y -391.465,Z 825.633,A 0.000,B 0.000,C 90.000,E1 149.999} C_DIS
LIN {X 0.082,Y -392.461,Z 825.632,A 0.000,B 0.000,C 90.000,E1 149.793} C_DIS
LIN {X 0.247,Y -395.698,Z 825.630,A 0.000,B 0.000,C 90.000,E1 149.331} C_DIS
LIN {X 0.209,Y -403.088,Z 825.626,A 0.000,B 0.000,C 90.000,E1 148.663} C_DIS
LIN {X 0.093,Y -405.117,Z 825.625,A 0.000,B 0.000,C 90.000,E1 148.535} C_DIS
LIN {X -0.259,Y -411.356,Z 825.623,A 0.000,B 0.000,C 90.000,E1 148.201} C_DIS
LIN {X 0.017,Y -414.827,Z 825.622,A 0.000,B 0.000,C 90.000,E1 147.946} C_DIS
LIN {X -0.235,Y -428.270,Z 825.618,A 0.000,B 0.000,C 90.000,E1 147.248} C_DIS
LIN {X 0.023,Y -434.532,Z 825.616,A 0.000,B 0.000,C 90.000,E1 146.834} C_DIS
LIN {X 0.085,Y -441.000,Z 825.614,A 0.000,B 0.000,C 90.000,E1 146.421} C_DIS
LIN {X 0.023,Y -444.004,Z 825.612,A 0.000,B 0.000,C 90.000,E1 146.215} C_DIS
LIN {X 0.127,Y -451.512,Z 825.609,A 0.000,B 0.000,C 90.000,E1 145.595} C_DIS
LIN {X -0.031,Y -460.316,Z 825.605,A 0.000,B 0.000,C 90.000,E1 144.815} C_DIS
LIN {X 0.012,Y -464.713,Z 825.602,A 0.000,B 0.000,C 90.000,E1 144.402} C_DIS
LIN {X -0.212,Y -471.141,Z 825.598,A 0.000,B 0.000,C 90.000,E1 143.703} C_DIS
LIN {X -0.166,Y -478.548,Z 825.593,A 0.000,B 0.000,C 90.000,E1 142.763} C_DIS
LIN {X -0.254,Y -487.693,Z 825.586,A 0.000,B 0.000,C 90.000,E1 141.537} C_DIS
LIN {X 0.098,Y -492.057,Z 825.583,A 0.000,B 0.000,C 90.000,E1 140.884} C_DIS
LIN {X -0.038,Y -498.296,Z 825.578,A 0.000,B 0.000,C 90.000,E1 139.989} C_DIS
LIN {X 0.101,Y -505.496,Z 825.571,A 0.000,B 0.000,C 90.000,E1 138.771} C_DIS
LIN {X -0.151,Y -511.404,Z 825.565,A 0.000,B 0.000,C 90.000,E1 137.757} C_DIS
LIN {X -0.085,Y -516.138,Z 825.560,A 0.000,B 0.000,C 90.000,E1 136.863} C_DIS
LIN {X -0.146,Y -523.746,Z 825.552,A 0.000,B 0.000,C 90.000,E1 135.405} C_DIS
LIN {X -0.019,Y -529.683,Z 825.546,A 0.000,B 0.000,C 90.000,E1 134.231} C_DIS
LIN {X 0.271,Y -532.513,Z 825.543,A 0.000,B 0.000,C 90.000,E1 133.623} C_DIS
LIN {X 0.363,Y -537.330,Z 825.537,A 0.000,B 0.000,C 90.000,E1 132.609} C_DIS
LIN {X 0.123,Y -543.038,Z 825.530,A 0.000,B 0.000,C 90.000,E1 131.353} C_DIS
LIN {X -0.215,Y -546.575,Z 825.525,A 0.000,B 0.000,C 90.000,E1 130.539} C_DIS
LIN {X 0.212,Y -548.819,Z 825.522,A 0.000,B 0.000,C 90.000,E1 129.930} C_DIS
LIN {X -0.010,Y -552.864,Z 825.516,A 0.000,B 0.000,C 90.000,E1 128.830} C_DIS
LIN {X -0.177,Y -556.466,Z 825.510,A 0.000,B 0.000,C 90.000,E1 127.729} C_DIS
LIN {X 0.150,Y -559.782,Z 825.503,A 0.000,B 0.000,C 90.000,E1 126.583} C_DIS
LIN {X 0.098,Y -561.676,Z 825.499,A 0.000,B 0.000,C 90.000,E1 125.758} C_DIS
LIN {X -0.065,Y -563.093,Z 825.494,A 0.000,B 0.000,C 90.000,E1 124.945} C_DIS
LIN {X -0.080,Y -564.206,Z 825.490,A 0.000,B 0.000,C 90.000,E1 124.119} C_DIS
LIN {X 0.023,Y -565.155,Z 825.483,A 0.000,B 0.000,C 90.000,E1 123.007} C_DIS
LIN {X -0.275,Y -565.757,Z 825.479,A 0.000,B 0.000,C 90.000,E1 122.212} C_DIS
LIN {X 0.116,Y -565.927,Z 825.476,A 0.000,B 0.000,C 90.000,E1 121.623} C_DIS
LIN {X 0.036,Y -565.933,Z 825.468,A 0.000,B 0.000,C 90.000,E1 120.256} C_DIS
LIN {X 0.245,Y -565.288,Z 825.464,A 0.000,B 0.000,C 90.000,E1 119.411} C_DIS
LIN {X 0.074,Y -564.022,Z 825.456,A 0.000,B 0.000,C 90.000,E1 118.052} C_DIS
LIN {X -0.041,Y -563.380,Z 825.453,A 0.000,B 0.000,C 90.000,E1 117.513} C_DIS
LIN {X -0.232,Y -562.947,Z 825.451,A 0.000,B 0.000,C 90.000,E1 117.257} C_DIS
LIN {X 0.078,Y -562.678,Z 825.450,A 0.000,B 0.000,C 90.000,E1 116.950} C_DIS
LIN {X 0.251,Y -561.388,Z 825.445,A 0.000,B 0.000,C 90.000,E1 116.104} C_DIS
LIN {X -0.144,Y -560.735,Z 825.442,A 0.000,B 0.000,C 90.000,E1 115.591} C_DIS
LIN {X 0.163,Y -560.299,Z 825.441,A 0.000,B 0.000,C 90.000,E1 115.283} C_DIS
LIN {X -0.037,Y -560.136,Z 825.439,A 0.000,B 0.000,C 90.000,E1 115.027} C_DIS
LIN {X -0.139,Y -559.893,Z 825.438,A 0.000,B 0.000,C 90.000,E1 114.899} C_DIS
LIN {X 0.125,Y -560.370,Z 825.432,A 0.000,B 0.000,C 90.000,E1 113.770} C_DIS
LIN {X -0.290,Y -561.604,Z 825.423,A 0.000,B 0.000,C 90.000,E1 112.153} C_DIS
LIN {X -0.276,Y -562.212,Z 825.417,A 0.000,B 0.000,C 90.000,E1 111.046} C_DIS
LIN {X -0.168,Y -562.381,Z 825.414,A 0.000,B 0.000,C 90.000,E1 110.482} C_DIS
LIN {X -0.340,Y -562.595,Z 825.408,A 0.000,B 0.000,C 90.000,E1 109.396} C_DIS
LIN {X 0.036,Y -562.637,Z 825.395,A 0.000,B 0.000,C 90.000,E1 107.149} C_DIS
LIN {X -0.021,Y -563.410,Z 825.378,A 0.000,B 0.000,C 90.000,E1 104.120} C_DIS
LIN {X 0.071,Y -563.954,Z 825.372,A 0.000,B 0.000,C 90.000,E1 103.008} C_DIS
LIN {X -0.260,Y -565.370,Z 825.360,A 0.000,B 0.000,C 90.000,E1 100.838} C_DIS
LIN {X -0.066,Y -566.423,Z 825.352,A 0.000,B 0.000,C 90.000,E1 99.443} C_DIS
LIN {X -0.244,Y -567.540,Z 825.343,A 0.000,B 0.000,C 90.000,E1 97.814} C_DIS
LIN {X 0.006,Y -568.521,Z 825.334,A 0.000,B 0.000,C 90.000,E1 96.144} C_DIS
LIN {X 0.280,Y -569.352,Z 825.325,A 0.000,B 0.000,C 90.000,E1 94.473} C_DIS
LIN {X -0.173,Y -569.928,Z 825.317,A 0.000,B 0.000,C 90.000,E1 93.151} C_DIS
LIN {X 0.173,Y -570.562,Z 825.307,A 0.000,B 0.000,C 90.000,E1 91.203} C_DIS
LIN {X 0.265,Y -570.940,Z 825.299,A 0.000,B 0.000,C 90.000,E1 89.828} C_DIS
LIN {X -0.077,Y -571.379,Z 825.290,A 0.000,B 0.000,C 90.000,E1 88.224} C_DIS
LIN {X -0.228,Y -571.591,Z 825.286,A 0.000,B 0.000,C 90.000,E1 87.421} C_DIS
LIN {X 0.061,Y -571.924,Z 825.276,A 0.000,B 0.000,C 90.000,E1 85.755} C_DIS
LIN {X 0.229,Y -572.169,Z 825.269,A 0.000,B 0.000,C 90.000,E1 84.375} C_DIS
LIN {X 0.201,Y -572.572,Z 825.258,A 0.000,B 0.000,C 90.000,E1 82.470} C_DIS
LIN {X 0.169,Y -573.043,Z 825.248,A 0.000,B 0.000,C 90.000,E1 80.566} C_DIS
LIN {X 0.232,Y -573.506,Z 825.239,A 0.000,B 0.000,C 90.000,E1 78.926} C_DIS
LIN {X -0.005,Y -573.841,Z 825.231,A 0.000,B 0.000,C 90.000,E1 77.589} C_DIS
LIN {X 0.009,Y -574.051,Z 825.224,A 0.000,B 0.000,C 90.000,E1 76.228} C_DIS
LIN {X 0.036,Y -574.224,Z 825.216,A 0.000,B 0.000,C 90.000,E1 74.866} C_DIS
LIN {X 0.059,Y -574.224,Z 825.208,A 0.000,B 0.000,C 90.000,E1 73.504} C_DIS
LIN {X 0.050,Y -574.168,Z 825.199,A 0.000,B 0.000,C 90.000,E1 71.873} C_DIS
LIN {X 0.222,Y -573.967,Z 825.192,A 0.000,B 0.000,C 90.000,E1 70.496} C_DIS
LIN {X -0.142,Y -573.664,Z 825.183,A 0.000,B 0.000,C 90.000,E1 68.901} C_DIS
LIN {X -0.128,Y -573.342,Z 825.175,A 0.000,B 0.000,C 90.000,E1 67.539} C_DIS
LIN {X -0.286,Y -572.768,Z 825.166,A 0.000,B 0.000,C 90.000,E1 65.921} C_DIS
LIN {X -0.064,Y -572.187,Z 825.159,A 0.000,B 0.000,C 90.000,E1 64.537} C_DIS
LIN {X -0.115,Y -571.519,Z 825.151,A 0.000,B 0.000,C 90.000,E1 63.179} C_DIS
LIN {X 0.334,Y -570.684,Z 825.143,A 0.000,B 0.000,C 90.000,E1 61.769} C_DIS
LIN {X -0.245,Y -569.557,Z 825.136,A 0.000,B 0.000,C 90.000,E1 60.461} C_DIS
LIN {X 0.110,Y -568.325,Z 825.130,A 0.000,B 0.000,C 90.000,E1 59.331} C_DIS
LIN {X -0.037,Y -567.011,Z 825.124,A 0.000,B 0.000,C 90.000,E1 58.250} C_DIS
LIN {X -0.200,Y -565.472,Z 825.118,A 0.000,B 0.000,C 90.000,E1 57.168} C_DIS
LIN {X 0.077,Y -563.694,Z 825.111,A 0.000,B 0.000,C 90.000,E1 56.040} C_DIS
LIN {X -0.296,Y -561.638,Z 825.105,A 0.000,B 0.000,C 90.000,E1 54.975} C_DIS
LIN {X 0.094,Y -559.198,Z 825.099,A 0.000,B 0.000,C 90.000,E1 53.829} C_DIS
LIN {X 0.031,Y -557.206,Z 825.095,A 0.000,B 0.000,C 90.000,E1 53.004} C_DIS
LIN {X -0.165,Y -554.926,Z 825.090,A 0.000,B 0.000,C 90.000,E1 52.190} C_DIS
LIN {X -0.015,Y -553.307,Z 825.087,A 0.000,B 0.000,C 90.000,E1 51.618} C_DIS
LIN {X -0.246,Y -550.559,Z 825.082,A 0.000,B 0.000,C 90.000,E1 50.803} C_DIS
LIN {X 0.269,Y -547.447,Z 825.077,A 0.000,B 0.000,C 90.000,E1 49.908} C_DIS
LIN {X -0.060,Y -545.294,Z 825.074,A 0.000,B 0.000,C 90.000,E1 49.380} C_DIS
LIN {X -0.212,Y -542.186,Z 825.070,A 0.000,B 0.000,C 90.000,E1 48.690} C_DIS
LIN {X 0.010,Y -538.816,Z 825.066,A 0.000,B 0.000,C 90.000,E1 47.957} C_DIS
LIN {X -0.021,Y -535.873,Z 825.063,A 0.000,B 0.000,C 90.000,E1 47.391} C_DIS
LIN {X -0.068,Y -532.627,Z 825.060,A 0.000,B 0.000,C 90.000,E1 46.824} C_DIS
LIN {X 0.248,Y -529.029,Z 825.057,A 0.000,B 0.000,C 90.000,E1 46.215} C_DIS
LIN {X -0.285,Y -524.209,Z 825.053,A 0.000,B 0.000,C 90.000,E1 45.567} C_DIS
LIN {X -0.041,Y -519.881,Z 825.050,A 0.000,B 0.000,C 90.000,E1 44.960} C_DIS
LIN {X 0.028,Y -516.421,Z 825.047,A 0.000,B 0.000,C 90.000,E1 44.514} C_DIS
LIN {X -0.150,Y -511.385,Z 825.044,A 0.000,B 0.000,C 90.000,E1 43.947} C_DIS
LIN {X 0.058,Y -506.063,Z 825.041,A 0.000,B 0.000,C 90.000,E1 43.338} C_DIS
LIN {X -0.068,Y -502.059,Z 825.039,A 0.000,B 0.000,C 90.000,E1 42.933} C_DIS
LIN {X -0.133,Y -493.601,Z 825.034,A 0.000,B 0.000,C 90.000,E1 42.123} C_DIS
LIN {X -0.130,Y -487.646,Z 825.031,A 0.000,B 0.000,C 90.000,E1 41.595} C_DIS
LIN {X 0.093,Y -481.489,Z 825.028,A 0.000,B 0.000,C 90.000,E1 41.067} C_DIS
LIN {X -0.200,Y -470.690,Z 825.024,A 0.000,B 0.000,C 90.000,E1 40.253} C_DIS
LIN {X 0.082,Y -459.629,Z 825.019,A 0.000,B 0.000,C 90.000,E1 39.402} C_DIS
LIN {X -0.190,Y -442.330,Z 825.012,A 0.000,B 0.000,C 90.000,E1 38.177} C_DIS
LIN {X 0.229,Y -418.908,Z 825.002,A 0.000,B 0.000,C 90.000,E1 36.297} C_DIS
LIN {X 0.209,Y -406.817,Z 824.996,A 0.000,B 0.000,C 90.000,E1 35.231} C_DIS
LIN {X -0.083,Y -401.040,Z 824.993,A 0.000,B 0.000,C 90.000,E1 34.692} C_DIS
LIN {X -0.044,Y -399.775,Z 824.992,A 0.000,B 0.000,C 90.000,E1 34.532} C_DIS
LIN {X -0.074,Y -397.370,Z 824.990,A 0.000,B 0.000,C 90.000,E1 34.199} C_DIS
LIN {X -0.112,Y -397.354,Z 824.990,A 0.000,B 0.000,C 90.000,E1 34.199} C_DIS
LIN {X 0.130,Y -393.881,Z 824.977,A 0.000,B 0.000,C 90.000,E1 31.878} C_DIS
LIN {X -0.008,Y -392.056,Z 824.972,A 0.000,B 0.000,C 90.000,E1 30.924} C_DIS
LIN {X 0.206,Y -393.771,Z 824.952,A 0.000,B 0.000,C 90.000,E1 27.257} C_DIS
LIN {X -0.090,Y -395.370,Z 824.938,A 0.000,B 0.000,C 90.000,E1 24.823} C_DIS
LIN {X -0.014,Y -396.955,Z 824.926,A 0.000,B 0.000,C 90.000,E1 22.695} C_DIS
LIN {X -0.125,Y -398.936,Z 824.912,A 0.000,B 0.000,C 90.000,E1 20.248} C_DIS
LIN {X -0.131,Y -402.241,Z 824.895,A 0.000,B 0.000,C 90.000,E1 17.094} C_DIS
LIN {X -0.087,Y -405.332,Z 824.881,A 0.000,B 0.000,C 90.000,E1 14.647} C_DIS
LIN {X 0.133,Y -408.526,Z 824.870,A 0.000,B 0.000,C 90.000,E1 12.535} C_DIS
LIN {X 0.064,Y -413.667,Z 824.853,A 0.000,B 0.000,C 90.000,E1 9.443} C_DIS
LIN {X -0.071,Y -417.342,Z 824.841,A 0.000,B 0.000,C 90.000,E1 7.409} C_DIS
LIN {X 0.056,Y -419.789,Z 824.834,A 0.000,B 0.000,C 90.000,E1 6.030} C_DIS
LIN {X -0.015,Y -424.160,Z 824.820,A 0.000,B 0.000,C 90.000,E1 3.669} C_DIS
LIN {X -0.090,Y -428.195,Z 824.809,A 0.000,B 0.000,C 90.000,E1 1.661} C_DIS
LIN {X -0.019,Y -434.446,Z 824.793,A 0.000,B 0.000,C 90.000,E1 358.797} C_DIS
LIN {X 0.160,Y -439.052,Z 824.782,A 0.000,B 0.000,C 90.000,E1 356.788} C_DIS
LIN {X -0.105,Y -443.121,Z 824.773,A 0.000,B 0.000,C 90.000,E1 355.179} C_DIS
LIN {X -0.126,Y -448.045,Z 824.762,A 0.000,B 0.000,C 90.000,E1 353.223} C_DIS
LIN {X -0.126,Y -452.458,Z 824.753,A 0.000,B 0.000,C 90.000,E1 351.602} C_DIS
LIN {X -0.235,Y -454.706,Z 824.750,A 0.000,B 0.000,C 90.000,E1 350.971} C_DIS
LIN {X -0.024,Y -456.170,Z 824.748,A 0.000,B 0.000,C 90.000,E1 350.622} C_DIS
LIN {X -0.104,Y -459.357,Z 824.745,A 0.000,B 0.000,C 90.000,E1 350.151} C_DIS
LIN {X -0.030,Y -460.673,Z 824.744,A 0.000,B 0.000,C 90.000,E1 349.982} C_DIS
LIN {X 0.199,Y -462.716,Z 824.743,A 0.000,B 0.000,C 90.000,E1 349.746} C_DIS
LIN {X -0.258,Y -468.437,Z 824.741,A 0.000,B 0.000,C 90.000,E1 349.342} C_DIS
LIN {X -0.049,Y -476.110,Z 824.738,A 0.000,B 0.000,C 90.000,E1 348.814} C_DIS
LIN {X -0.081,Y -487.530,Z 824.734,A 0.000,B 0.000,C 90.000,E1 348.105} C_DIS
LIN {X -0.008,Y -503.518,Z 824.728,A 0.000,B 0.000,C 90.000,E1 347.061} C_DIS
LIN {X 0.227,Y -512.865,Z 824.725,A 0.000,B 0.000,C 90.000,E1 346.408} C_DIS
LIN {X -0.059,Y -525.360,Z 824.720,A 0.000,B 0.000,C 90.000,E1 345.574} C_DIS
LIN {X -0.242,Y -534.385,Z 824.716,A 0.000,B 0.000,C 90.000,E1 344.936} C_DIS
LIN {X 0.127,Y -543.288,Z 824.712,A 0.000,B 0.000,C 90.000,E1 344.212} C_DIS
LIN {X 0.201,Y -550.453,Z 824.709,A 0.000,B 0.000,C 90.000,E1 343.614} C_DIS
LIN {X -0.027,Y -558.680,Z 824.705,A 0.000,B 0.000,C 90.000,E1 342.906} C_DIS
LIN {X -0.173,Y -563.945,Z 824.702,A 0.000,B 0.000,C 90.000,E1 342.417} C_DIS
LIN {X -0.204,Y -570.258,Z 824.699,A 0.000,B 0.000,C 90.000,E1 341.764} C_DIS
LIN {X 0.007,Y -575.076,Z 824.696,A 0.000,B 0.000,C 90.000,E1 341.221} C_DIS
LIN {X 0.288,Y -578.638,Z 824.693,A 0.000,B 0.000,C 90.000,E1 340.786} C_DIS
LIN {X -0.029,Y -585.072,Z 824.689,A 0.000,B 0.000,C 90.000,E1 340.007} C_DIS
LIN {X -0.025,Y -589.967,Z 824.685,A 0.000,B 0.000,C 90.000,E1 339.337} C_DIS
LIN {X 0.237,Y -594.439,Z 824.682,A 0.000,B 0.000,C 90.000,E1 338.646} C_DIS
LIN {X 0.281,Y -599.387,Z 824.677,A 0.000,B 0.000,C 90.000,E1 337.847} C_DIS
LIN {X -0.219,Y -604.917,Z 824.672,A 0.000,B 0.000,C 90.000,E1 336.975} C_DIS
LIN {X -0.145,Y -611.744,Z 824.665,A 0.000,B 0.000,C 90.000,E1 335.793} C_DIS
LIN {X 0.305,Y -616.838,Z 824.660,A 0.000,B 0.000,C 90.000,E1 334.845} C_DIS
LIN {X -0.012,Y -622.250,Z 824.655,A 0.000,B 0.000,C 90.000,E1 333.845} C_DIS
LIN {X 0.007,Y -627.315,Z 824.649,A 0.000,B 0.000,C 90.000,E1 332.820} C_DIS
LIN {X 0.358,Y -630.840,Z 824.645,A 0.000,B 0.000,C 90.000,E1 332.025} C_DIS
LIN {X -0.031,Y -636.509,Z 824.638,A 0.000,B 0.000,C 90.000,E1 330.795} C_DIS
LIN {X -0.078,Y -640.901,Z 824.632,A 0.000,B 0.000,C 90.000,E1 329.793} C_DIS
LIN {X -0.061,Y -644.964,Z 824.627,A 0.000,B 0.000,C 90.000,E1 328.791} C_DIS
LIN {X 0.007,Y -648.680,Z 824.621,A 0.000,B 0.000,C 90.000,E1 327.788} C_DIS
LIN {X 0.118,Y -652.174,Z 824.616,A 0.000,B 0.000,C 90.000,E1 326.786} C_DIS
LIN {X 0.088,Y -656.945,Z 824.607,A 0.000,B 0.000,C 90.000,E1 325.308} C_DIS
LIN {X 0.219,Y -660.451,Z 824.601,A 0.000,B 0.000,C 90.000,E1 324.069} C_DIS
LIN {X 0.255,Y -663.621,Z 824.594,A 0.000,B 0.000,C 90.000,E1 322.844} C_DIS
LIN {X 0.345,Y -666.489,Z 824.587,A 0.000,B 0.000,C 90.000,E1 321.618} C_DIS
LIN {X -0.121,Y -668.009,Z 824.583,A 0.000,B 0.000,C 90.000,E1 320.928} C_DIS
LIN {X 0.029,Y -670.425,Z 824.576,A 0.000,B 0.000,C 90.000,E1 319.703} C_DIS
LIN {X 0.131,Y -672.593,Z 824.569,A 0.000,B 0.000,C 90.000,E1 318.485} C_DIS
LIN {X -0.254,Y -674.338,Z 824.564,A 0.000,B 0.000,C 90.000,E1 317.553} C_DIS
LIN {X -0.181,Y -675.483,Z 824.560,A 0.000,B 0.000,C 90.000,E1 316.824} C_DIS
LIN {X 0.019,Y -677.454,Z 824.552,A 0.000,B 0.000,C 90.000,E1 315.364} C_DIS
LIN {X 0.088,Y -678.122,Z 824.549,A 0.000,B 0.000,C 90.000,E1 314.879} C_DIS
LIN {X -0.072,Y -680.315,Z 824.539,A 0.000,B 0.000,C 90.000,E1 312.975} C_DIS
LIN {X 0.230,Y -681.956,Z 824.531,A 0.000,B 0.000,C 90.000,E1 311.515} C_DIS
LIN {X 0.076,Y -683.255,Z 824.524,A 0.000,B 0.000,C 90.000,E1 310.334} C_DIS
LIN {X 0.386,Y -684.400,Z 824.518,A 0.000,B 0.000,C 90.000,E1 309.116} C_DIS
LIN {X -0.110,Y -685.636,Z 824.510,A 0.000,B 0.000,C 90.000,E1 307.729} C_DIS
LIN {X -0.039,Y -686.882,Z 824.502,A 0.000,B 0.000,C 90.000,E1 306.297} C_DIS
LIN {X 0.023,Y -687.809,Z 824.495,A 0.000,B 0.000,C 90.000,E1 305.105} C_DIS
LIN {X 0.098,Y -688.663,Z 824.489,A 0.000,B 0.000,C 90.000,E1 303.913} C_DIS
LIN {X 0.243,Y -690.058,Z 824.478,A 0.000,B 0.000,C 90.000,E1 302.005} C_DIS
LIN {X 0.189,Y -691.073,Z 824.470,A 0.000,B 0.000,C 90.000,E1 300.590} C_DIS
LIN {X -0.198,Y -692.087,Z 824.462,A 0.000,B 0.000,C 90.000,E1 299.205} C_DIS
LIN {X 0.281,Y -693.272,Z 824.453,A 0.000,B 0.000,C 90.000,E1 297.513} C_DIS
LIN {X -0.153,Y -694.610,Z 824.444,A 0.000,B 0.000,C 90.000,E1 295.899} C_DIS
LIN {X 0.139,Y -695.777,Z 824.436,A 0.000,B 0.000,C 90.000,E1 294.463} C_DIS
LIN {X 0.012,Y -695.914,Z 824.433,A 0.000,B 0.000,C 90.000,E1 294.003} C_DIS
LIN {X -0.017,Y -695.934,Z 824.432,A 0.000,B 0.000,C 90.000,E1 293.770} C_DIS
LIN {X 0.236,Y -695.603,Z 824.431,A 0.000,B 0.000,C 90.000,E1 293.515} C_DIS
LIN {X -0.176,Y -694.628,Z 824.428,A 0.000,B 0.000,C 90.000,E1 293.078} C_DIS
LIN {X 0.071,Y -693.420,Z 824.427,A 0.000,B 0.000,C 90.000,E1 292.823} C_DIS
LIN {X 0.283,Y -689.561,Z 824.424,A 0.000,B 0.000,C 90.000,E1 292.333} C_DIS
LIN {X 0.398,Y -688.274,Z 824.424,A 0.000,B 0.000,C 90.000,E1 292.206} C_DIS
LIN {X -0.385,Y -686.310,Z 824.423,A 0.000,B 0.000,C 90.000,E1 292.153} C_DIS
LIN {X 0.209,Y -681.093,Z 824.422,A 0.000,B 0.000,C 90.000,E1 291.844} C_DIS
LIN {X 0.156,Y -679.212,Z 824.421,A 0.000,B 0.000,C 90.000,E1 291.770} C_DIS
LIN {X 0.076,Y -672.754,Z 824.420,A 0.000,B 0.000,C 90.000,E1 291.589} C_DIS
LIN {X 0.125,Y -670.685,Z 824.420,A 0.000,B 0.000,C 90.000,E1 291.535} C_DIS
LIN {X -0.177,Y -662.026,Z 824.419,A 0.000,B 0.000,C 90.000,E1 291.408} C_DIS
LIN {X 0.084,Y -647.997,Z 824.418,A 0.000,B 0.000,C 90.000,E1 291.153} C_DIS
LIN {X -0.130,Y -637.747,Z 824.417,A 0.000,B 0.000,C 90.000,E1 290.972} C_DIS
LIN {X 0.280,Y -627.024,Z 824.415,A 0.000,B 0.000,C 90.000,E1 290.663} C_DIS
LIN {X 0.290,Y -622.201,Z 824.414,A 0.000,B 0.000,C 90.000,E1 290.482} C_DIS
LIN {X 0.152,Y -620.124,Z 824.414,A 0.000,B 0.000,C 90.000,E1 290.429} C_DIS
LIN {X 0.125,Y -614.108,Z 824.412,A 0.000,B 0.000,C 90.000,E1 290.120} C_DIS
LIN {X -0.252,Y -612.348,Z 824.411,A 0.000,B 0.000,C 90.000,E1 289.993} C_DIS
LIN {X 0.265,Y -612.294,Z 824.411,A 0.000,B 0.000,C 90.000,E1 289.939} C_DIS
LIN {X 0.292,Y -612.019,Z 824.410,A 0.000,B 0.000,C 90.000,E1 289.758} C_DIS
LIN {X 0.267,Y -612.214,Z 824.409,A 0.000,B 0.000,C 90.000,E1 289.631} C_DIS
LIN {X -0.008,Y -614.137,Z 824.406,A 0.000,B 0.000,C 90.000,E1 289.141} C_DIS
LIN {X -0.242,Y -621.783,Z 824.399,A 0.000,B 0.000,C 90.000,E1 287.873} C_DIS
LIN {X 0.109,Y -623.665,Z 824.397,A 0.000,B 0.000,C 90.000,E1 287.457} C_DIS
LIN {X -0.141,Y -626.019,Z 824.394,A 0.000,B 0.000,C 90.000,E1 286.968} C_DIS
LIN {X -0.163,Y -628.976,Z 824.390,A 0.000,B 0.000,C 90.000,E1 286.205} C_DIS
LIN {X 0.219,Y -630.687,Z 824.387,A 0.000,B 0.000,C 90.000,E1 285.662} C_DIS
LIN {X -0.165,Y -632.203,Z 824.384,A 0.000,B 0.000,C 90.000,E1 285.190} C_DIS
LIN {X 0.074,Y -633.380,Z 824.382,A 0.000,B 0.000,C 90.000,E1 284.662} C_DIS
LIN {X 0.301,Y -634.814,Z 824.377,A 0.000,B 0.000,C 90.000,E1 283.883} C_DIS
LIN {X -0.056,Y -635.398,Z 824.375,A 0.000,B 0.000,C 90.000,E1 283.411} C_DIS
LIN {X 0.209,Y -635.704,Z 824.372,A 0.000,B 0.000,C 90.000,E1 282.883} C_DIS
LIN {X 0.033,Y -635.809,Z 824.370,A 0.000,B 0.000,C 90.000,E1 282.647} C_DIS
LIN {X 0.125,Y -635.434,Z 824.366,A 0.000,B 0.000,C 90.000,E1 281.883} C_DIS
LIN {X -0.182,Y -635.223,Z 824.365,A 0.000,B 0.000,C 90.000,E1 281.658} C_DIS
LIN {X -0.095,Y -633.996,Z 824.361,A 0.000,B 0.000,C 90.000,E1 280.894} C_DIS
LIN {X 0.160,Y -632.771,Z 824.358,A 0.000,B 0.000,C 90.000,E1 280.366} C_DIS
LIN {X -0.328,Y -631.097,Z 824.355,A 0.000,B 0.000,C 90.000,E1 279.905} C_DIS
LIN {X -0.096,Y -629.137,Z 824.352,A 0.000,B 0.000,C 90.000,E1 279.378} C_DIS
LIN {X 0.171,Y -627.406,Z 824.350,A 0.000,B 0.000,C 90.000,E1 278.973} C_DIS
LIN {X -0.190,Y -625.468,Z 824.348,A 0.000,B 0.000,C 90.000,E1 278.624} C_DIS
LIN {X -0.099,Y -622.444,Z 824.345,A 0.000,B 0.000,C 90.000,E1 278.106} C_DIS
LIN {X -0.027,Y -618.754,Z 824.342,A 0.000,B 0.000,C 90.000,E1 277.587} C_DIS
LIN {X 0.022,Y -614.251,Z 824.339,A 0.000,B 0.000,C 90.000,E1 277.068} C_DIS
LIN {X -0.231,Y -611.516,Z 824.338,A 0.000,B 0.000,C 90.000,E1 276.834} C_DIS
LIN {X 0.310,Y -607.542,Z 824.336,A 0.000,B 0.000,C 90.000,E1 276.429} C_DIS
LIN {X -0.069,Y -602.472,Z 824.334,A 0.000,B 0.000,C 90.000,E1 276.144} C_DIS
LIN {X 0.031,Y -597.710,Z 824.333,A 0.000,B 0.000,C 90.000,E1 275.853} C_DIS
LIN {X -0.263,Y -592.480,Z 824.331,A 0.000,B 0.000,C 90.000,E1 275.625} C_DIS
LIN {X -0.218,Y -587.337,Z 824.330,A 0.000,B 0.000,C 90.000,E1 275.391} C_DIS
LIN {X -0.102,Y -580.071,Z 824.328,A 0.000,B 0.000,C 90.000,E1 275.106} C_DIS
LIN {X -0.084,Y -574.432,Z 824.327,A 0.000,B 0.000,C 90.000,E1 274.935} C_DIS
LIN {X -0.035,Y -572.425,Z 824.327,A 0.000,B 0.000,C 90.000,E1 274.878} C_DIS
LIN {X 0.157,Y -566.488,Z 824.327,A 0.000,B 0.000,C 90.000,E1 274.759} C_DIS
LIN {X 0.011,Y -559.921,Z 824.326,A 0.000,B 0.000,C 90.000,E1 274.759} C_DIS
LIN {X -0.036,Y -552.143,Z 824.326,A 0.000,B 0.000,C 90.000,E1 274.759} C_DIS
LIN {X -0.214,Y -551.567,Z 824.326,A 0.000,B 0.000,C 90.000,E1 274.759} C_DIS
LIN {X -0.177,Y -550.116,Z 824.325,A 0.000,B 0.000,C 90.000,E1 274.588} C_DIS
LIN {X -0.219,Y -550.088,Z 824.325,A 0.000,B 0.000,C 90.000,E1 274.588} C_DIS
LIN {X -0.003,Y -549.734,Z 824.325,A 0.000,B 0.000,C 90.000,E1 274.416} C_DIS
LIN {X 0.181,Y -548.750,Z 824.320,A 0.000,B 0.000,C 90.000,E1 273.555} C_DIS
LIN {X -0.100,Y -547.696,Z 824.312,A 0.000,B 0.000,C 90.000,E1 272.178} C_DIS
LIN {X 0.189,Y -546.476,Z 824.303,A 0.000,B 0.000,C 90.000,E1 270.458} C_DIS
LIN {X -0.069,Y -545.081,Z 824.292,A 0.000,B 0.000,C 90.000,E1 268.511} C_DIS
LIN {X 0.243,Y -543.544,Z 824.279,A 0.000,B 0.000,C 90.000,E1 266.216} C_DIS
LIN {X -0.117,Y -542.843,Z 824.273,A 0.000,B 0.000,C 90.000,E1 265.122} C_DIS
LIN {X 0.071,Y -541.882,Z 824.265,A 0.000,B 0.000,C 90.000,E1 263.685} C_DIS
LIN {X -0.241,Y -540.692,Z 824.257,A 0.000,B 0.000,C 90.000,E1 262.299} C_DIS
LIN {X 0.109,Y -539.098,Z 824.248,A 0.000,B 0.000,C 90.000,E1 260.557} C_DIS
LIN {X -0.172,Y -537.696,Z 824.240,A 0.000,B 0.000,C 90.000,E1 259.162} C_DIS
LIN {X 0.145,Y -536.268,Z 824.232,A 0.000,B 0.000,C 90.000,E1 257.701} C_DIS
LIN {X -0.148,Y -535.179,Z 824.225,A 0.000,B 0.000,C 90.000,E1 256.589} C_DIS
LIN {X -0.062,Y -532.889,Z 824.214,A 0.000,B 0.000,C 90.000,E1 254.574} C_DIS
LIN {X -0.072,Y -530.934,Z 824.205,A 0.000,B 0.000,C 90.000,E1 252.851} C_DIS
LIN {X -0.005,Y -529.510,Z 824.198,A 0.000,B 0.000,C 90.000,E1 251.692} C_DIS
LIN {X 0.056,Y -527.653,Z 824.190,A 0.000,B 0.000,C 90.000,E1 250.242} C_DIS
LIN {X 0.257,Y -525.663,Z 824.182,A 0.000,B 0.000,C 90.000,E1 248.773} C_DIS
LIN {X -0.228,Y -522.793,Z 824.171,A 0.000,B 0.000,C 90.000,E1 246.794} C_DIS
LIN {X 0.067,Y -520.510,Z 824.163,A 0.000,B 0.000,C 90.000,E1 245.305} C_DIS
LIN {X -0.045,Y -517.642,Z 824.153,A 0.000,B 0.000,C 90.000,E1 243.563} C_DIS
LIN {X -0.107,Y -515.091,Z 824.145,A 0.000,B 0.000,C 90.000,E1 242.103} C_DIS
LIN {X 0.262,Y -512.395,Z 824.137,A 0.000,B 0.000,C 90.000,E1 240.589} C_DIS
LIN {X -0.222,Y -509.187,Z 824.127,A 0.000,B 0.000,C 90.000,E1 238.869} C_DIS
LIN {X -0.034,Y -506.849,Z 824.120,A 0.000,B 0.000,C 90.000,E1 237.661} C_DIS
LIN {X 0.183,Y -505.660,Z 824.117,A 0.000,B 0.000,C 90.000,E1 237.041} C_DIS
LIN {X 0.077,Y -501.755,Z 824.107,A 0.000,B 0.000,C 90.000,E1 235.261} C_DIS
LIN {X -0.247,Y -497.603,Z 824.097,A 0.000,B 0.000,C 90.000,E1 233.497} C_DIS
LIN {X -0.058,Y -493.255,Z 824.087,A 0.000,B 0.000,C 90.000,E1 231.662} C_DIS
LIN {X 0.039,Y -490.304,Z 824.080,A 0.000,B 0.000,C 90.000,E1 230.436} C_DIS
LIN {X -0.174,Y -485.321,Z 824.068,A 0.000,B 0.000,C 90.000,E1 228.324} C_DIS
LIN {X -0.002,Y -481.104,Z 824.058,A 0.000,B 0.000,C 90.000,E1 226.458} C_DIS
LIN {X 0.174,Y -476.503,Z 824.046,A 0.000,B 0.000,C 90.000,E1 224.271} C_DIS
LIN {X 0.103,Y -470.435,Z 824.031,A 0.000,B 0.000,C 90.000,E1 221.472} C_DIS
LIN {X 0.104,Y -465.187,Z 824.017,A 0.000,B 0.000,C 90.000,E1 218.955} C_DIS
LIN {X -0.219,Y -462.471,Z 824.010,A 0.000,B 0.000,C 90.000,E1 217.729} C_DIS
LIN {X 0.179,Y -459.209,Z 824.001,A 0.000,B 0.000,C 90.000,E1 216.091} C_DIS
LIN {X -0.130,Y -455.924,Z 823.992,A 0.000,B 0.000,C 90.000,E1 214.532} C_DIS
LIN {X 0.134,Y -450.527,Z 823.978,A 0.000,B 0.000,C 90.000,E1 211.926} C_DIS
LIN {X -0.002,Y -446.508,Z 823.967,A 0.000,B 0.000,C 90.000,E1 210.001} C_DIS
LIN {X 0.103,Y -443.339,Z 823.958,A 0.000,B 0.000,C 90.000,E1 208.359} C_DIS
LIN {X -0.029,Y -439.453,Z 823.947,A 0.000,B 0.000,C 90.000,E1 206.411} C_DIS
LIN {X 0.092,Y -436.842,Z 823.939,A 0.000,B 0.000,C 90.000,E1 205.079} C_DIS
LIN {X 0.214,Y -432.805,Z 823.928,A 0.000,B 0.000,C 90.000,E1 203.078} C_DIS
LIN {X -0.115,Y -428.301,Z 823.915,A 0.000,B 0.000,C 90.000,E1 200.791} C_DIS
LIN {X -0.102,Y -425.757,Z 823.908,A 0.000,B 0.000,C 90.000,E1 199.450} C_DIS
LIN {X 0.106,Y -421.768,Z 823.897,A 0.000,B 0.000,C 90.000,E1 197.402} C_DIS
LIN {X -0.150,Y -417.178,Z 823.884,A 0.000,B 0.000,C 90.000,E1 195.064} C_DIS
LIN {X -0.165,Y -414.658,Z 823.876,A 0.000,B 0.000,C 90.000,E1 193.703} C_DIS
LIN {X 0.123,Y -411.365,Z 823.867,A 0.000,B 0.000,C 90.000,E1 191.951} C_DIS
LIN {X -0.053,Y -408.055,Z 823.857,A 0.000,B 0.000,C 90.000,E1 190.254} C_DIS
LIN {X 0.031,Y -404.799,Z 823.847,A 0.000,B 0.000,C 90.000,E1 188.511} C_DIS
LIN {X -0.073,Y -400.310,Z 823.834,A 0.000,B 0.000,C 90.000,E1 186.087} C_DIS
LIN {X 0.136,Y -393.374,Z 823.810,A 0.000,B 0.000,C 90.000,E1 181.835} C_DIS
LIN {X 0.132,Y -388.756,Z 823.791,A 0.000,B 0.000,C 90.000,E1 178.282} C_DIS
LIN {X -0.130,Y -387.438,Z 823.785,A 0.000,B 0.000,C 90.000,E1 177.249} C_DIS
LIN {X -0.010,Y -384.489,Z 823.771,A 0.000,B 0.000,C 90.000,E1 174.723} C_DIS
LIN {X -0.167,Y -380.556,Z 823.751,A 0.000,B 0.000,C 90.000,E1 171.141} C_DIS
LIN {X -0.099,Y -377.885,Z 823.735,A 0.000,B 0.000,C 90.000,E1 168.229} C_DIS
LIN {X 0.115,Y -375.441,Z 823.718,A 0.000,B 0.000,C 90.000,E1 165.283} C_DIS
LIN {X -0.081,Y -373.127,Z 823.690,A 0.000,B 0.000,C 90.000,E1 160.188} C_DIS
LIN {X 0.000,Y -373.284,Z 823.678,A 0.000,B 0.000,C 90.000,E1 157.975} C_DIS
LIN {X 0.151,Y -373.845,Z 823.670,A 0.000,B 0.000,C 90.000,E1 156.485} C_DIS
LIN {X 0.005,Y -374.804,Z 823.663,A 0.000,B 0.000,C 90.000,E1 155.409} C_DIS
LIN {X -0.001,Y -376.733,Z 823.655,A 0.000,B 0.000,C 90.000,E1 153.948} C_DIS
LIN {X 0.091,Y -377.890,Z 823.651,A 0.000,B 0.000,C 90.000,E1 153.204} C_DIS
LIN {X -0.072,Y -378.775,Z 823.649,A 0.000,B 0.000,C 90.000,E1 152.871} C_DIS
LIN {X 0.065,Y -379.515,Z 823.647,A 0.000,B 0.000,C 90.000,E1 152.487} C_DIS
LIN {X -0.006,Y -381.895,Z 823.642,A 0.000,B 0.000,C 90.000,E1 151.591} C_DIS
LIN {X -0.025,Y -383.801,Z 823.639,A 0.000,B 0.000,C 90.000,E1 151.051} C_DIS
LIN {X 0.132,Y -384.943,Z 823.637,A 0.000,B 0.000,C 90.000,E1 150.667} C_DIS
LIN {X 0.083,Y -386.812,Z 823.635,A 0.000,B 0.000,C 90.000,E1 150.255} C_DIS
LIN {X 0.137,Y -390.031,Z 823.632,A 0.000,B 0.000,C 90.000,E1 149.665} C_DIS
LIN {X -0.098,Y -394.277,Z 823.628,A 0.000,B 0.000,C 90.000,E1 149.076} C_DIS
LIN {X -0.067,Y -397.957,Z 823.626,A 0.000,B 0.000,C 90.000,E1 148.614} C_DIS
LIN {X -0.156,Y -399.647,Z 823.625,A 0.000,B 0.000,C 90.000,E1 148.456} C_DIS
LIN {X -0.014,Y -408.143,Z 823.621,A 0.000,B 0.000,C 90.000,E1 147.740} C_DIS
LIN {X 0.161,Y -424.458,Z 823.615,A 0.000,B 0.000,C 90.000,E1 146.707} C_DIS
LIN {X -0.007,Y -436.344,Z 823.611,A 0.000,B 0.000,C 90.000,E1 146.008} C_DIS
LIN {X -0.101,Y -442.551,Z 823.609,A 0.000,B 0.000,C 90.000,E1 145.595} C_DIS
LIN {X 0.171,Y -450.149,Z 823.606,A 0.000,B 0.000,C 90.000,E1 144.975} C_DIS
LIN {X 0.046,Y -455.813,Z 823.603,A 0.000,B 0.000,C 90.000,E1 144.482} C_DIS
LIN {X 0.120,Y -460.119,Z 823.601,A 0.000,B 0.000,C 90.000,E1 144.069} C_DIS
LIN {X 0.234,Y -466.754,Z 823.596,A 0.000,B 0.000,C 90.000,E1 143.336} C_DIS
LIN {X -0.146,Y -470.641,Z 823.594,A 0.000,B 0.000,C 90.000,E1 142.924} C_DIS
LIN {X -0.111,Y -477.875,Z 823.589,A 0.000,B 0.000,C 90.000,E1 141.984} C_DIS
LIN {X -0.153,Y -487.986,Z 823.581,A 0.000,B 0.000,C 90.000,E1 140.598} C_DIS
LIN {X -0.018,Y -494.432,Z 823.576,A 0.000,B 0.000,C 90.000,E1 139.666} C_DIS
LIN {X -0.130,Y -500.074,Z 823.571,A 0.000,B 0.000,C 90.000,E1 138.771} C_DIS
LIN {X -0.163,Y -502.695,Z 823.568,A 0.000,B 0.000,C 90.000,E1 138.324} C_DIS
LIN {X -0.220,Y -510.180,Z 823.561,A 0.000,B 0.000,C 90.000,E1 136.986} C_DIS
LIN {X 0.314,Y -515.590,Z 823.555,A 0.000,B 0.000,C 90.000,E1 135.891} C_DIS
LIN {X -0.187,Y -520.875,Z 823.549,A 0.000,B 0.000,C 90.000,E1 134.919} C_DIS
LIN {X -0.038,Y -525.142,Z 823.545,A 0.000,B 0.000,C 90.000,E1 134.028} C_DIS
LIN {X -0.042,Y -530.273,Z 823.539,A 0.000,B 0.000,C 90.000,E1 133.014} C_DIS
LIN {X 0.193,Y -535.592,Z 823.533,A 0.000,B 0.000,C 90.000,E1 131.838} C_DIS
LIN {X 0.322,Y -540.918,Z 823.525,A 0.000,B 0.000,C 90.000,E1 130.539} C_DIS
LIN {X -0.008,Y -545.260,Z 823.519,A 0.000,B 0.000,C 90.000,E1 129.439} C_DIS
LIN {X -0.017,Y -547.192,Z 823.516,A 0.000,B 0.000,C 90.000,E1 128.874} C_DIS
LIN {X 0.115,Y -549.900,Z 823.511,A 0.000,B 0.000,C 90.000,E1 128.016} C_DIS
LIN {X 0.344,Y -553.248,Z 823.505,A 0.000,B 0.000,C 90.000,E1 126.870} C_DIS
LIN {X -0.226,Y -555.533,Z 823.500,A 0.000,B 0.000,C 90.000,E1 126.091} C_DIS
LIN {X 0.000,Y -557.085,Z 823.496,A 0.000,B 0.000,C 90.000,E1 125.231} C_DIS
LIN {X -0.078,Y -558.035,Z 823.491,A 0.000,B 0.000,C 90.000,E1 124.405} C_DIS
LIN {X -0.060,Y -558.955,Z 823.485,A 0.000,B 0.000,C 90.000,E1 123.293} C_DIS
LIN {X -0.119,Y -559.465,Z 823.480,A 0.000,B 0.000,C 90.000,E1 122.467} C_DIS
LIN {X 0.220,Y -559.647,Z 823.477,A 0.000,B 0.000,C 90.000,E1 121.878} C_DIS
LIN {X -0.257,Y -559.419,Z 823.470,A 0.000,B 0.000,C 90.000,E1 120.541} C_DIS
LIN {X -0.047,Y -558.932,Z 823.463,A 0.000,B 0.000,C 90.000,E1 119.411} C_DIS
LIN {X 0.090,Y -558.450,Z 823.459,A 0.000,B 0.000,C 90.000,E1 118.565} C_DIS
LIN {X 0.223,Y -558.127,Z 823.454,A 0.000,B 0.000,C 90.000,E1 117.719} C_DIS
LIN {X 0.015,Y -557.913,Z 823.453,A 0.000,B 0.000,C 90.000,E1 117.462} C_DIS
LIN {X 0.172,Y -557.887,Z 823.449,A 0.000,B 0.000,C 90.000,E1 116.821} C_DIS
LIN {X 0.141,Y -558.234,Z 823.448,A 0.000,B 0.000,C 90.000,E1 116.616} C_DIS
LIN {X -0.068,Y -558.263,Z 823.446,A 0.000,B 0.000,C 90.000,E1 116.360} C_DIS
LIN {X -0.276,Y -558.119,Z 823.445,A 0.000,B 0.000,C 90.000,E1 116.104} C_DIS
LIN {X 0.018,Y -558.520,Z 823.443,A 0.000,B 0.000,C 90.000,E1 115.796} C_DIS
LIN {X 0.347,Y -558.705,Z 823.440,A 0.000,B 0.000,C 90.000,E1 115.207} C_DIS
LIN {X 0.138,Y -558.990,Z 823.439,A 0.000,B 0.000,C 90.000,E1 114.951} C_DIS
LIN {X -0.004,Y -560.562,Z 823.428,A 0.000,B 0.000,C 90.000,E1 113.025} C_DIS
LIN {X 0.207,Y -561.431,Z 823.422,A 0.000,B 0.000,C 90.000,E1 111.897} C_DIS
LIN {X 0.216,Y -562.138,Z 823.416,A 0.000,B 0.000,C 90.000,E1 110.791} C_DIS
LIN {X 0.040,Y -562.591,Z 823.410,A 0.000,B 0.000,C 90.000,E1 109.704} C_DIS
LIN {X -0.025,Y -562.691,Z 823.400,A 0.000,B 0.000,C 90.000,E1 108.055} C_DIS
LIN {X -0.077,Y -563.172,Z 823.385,A 0.000,B 0.000,C 90.000,E1 105.300} C_DIS
LIN {X 0.232,Y -564.167,Z 823.373,A 0.000,B 0.000,C 90.000,E1 103.063} C_DIS
LIN {X -0.098,Y -565.531,Z 823.361,A 0.000,B 0.000,C 90.000,E1 100.894} C_DIS
LIN {X 0.269,Y -566.777,Z 823.351,A 0.000,B 0.000,C 90.000,E1 99.208} C_DIS
LIN {X 0.015,Y -567.904,Z 823.342,A 0.000,B 0.000,C 90.000,E1 97.587} C_DIS
LIN {X -0.225,Y -568.870,Z 823.333,A 0.000,B 0.000,C 90.000,E1 95.967} C_DIS
LIN {X 0.002,Y -569.675,Z 823.324,A 0.000,B 0.000,C 90.000,E1 94.302} C_DIS
LIN {X 0.125,Y -570.220,Z 823.316,A 0.000,B 0.000,C 90.000,E1 92.922} C_DIS
LIN {X -0.088,Y -570.886,Z 823.306,A 0.000,B 0.000,C 90.000,E1 91.031} C_DIS
LIN {X 0.009,Y -571.246,Z 823.298,A 0.000,B 0.000,C 90.000,E1 89.656} C_DIS
LIN {X 0.263,Y -571.699,Z 823.289,A 0.000,B 0.000,C 90.000,E1 87.993} C_DIS
LIN {X 0.096,Y -571.906,Z 823.284,A 0.000,B 0.000,C 90.000,E1 87.192} C_DIS
LIN {X -0.182,Y -572.236,Z 823.275,A 0.000,B 0.000,C 90.000,E1 85.584} C_DIS
LIN {X -0.013,Y -572.464,Z 823.268,A 0.000,B 0.000,C 90.000,E1 84.204} C_DIS
LIN {X -0.040,Y -572.879,Z 823.257,A 0.000,B 0.000,C 90.000,E1 82.299} C_DIS
LIN {X 0.022,Y -573.374,Z 823.247,A 0.000,B 0.000,C 90.000,E1 80.387} C_DIS
LIN {X -0.012,Y -573.797,Z 823.238,A 0.000,B 0.000,C 90.000,E1 78.757} C_DIS
LIN {X -0.130,Y -574.114,Z 823.230,A 0.000,B 0.000,C 90.000,E1 77.409} C_DIS
LIN {X 0.114,Y -574.262,Z 823.224,A 0.000,B 0.000,C 90.000,E1 76.297} C_DIS
LIN {X -0.073,Y -574.433,Z 823.215,A 0.000,B 0.000,C 90.000,E1 74.685} C_DIS
LIN {X -0.045,Y -574.394,Z 823.207,A 0.000,B 0.000,C 90.000,E1 73.323} C_DIS
LIN {X 0.136,Y -574.339,Z 823.200,A 0.000,B 0.000,C 90.000,E1 71.945} C_DIS
LIN {X 0.125,Y -574.083,Z 823.191,A 0.000,B 0.000,C 90.000,E1 70.315} C_DIS
LIN {X -0.239,Y -573.740,Z 823.182,A 0.000,B 0.000,C 90.000,E1 68.720} C_DIS
LIN {X -0.226,Y -573.363,Z 823.174,A 0.000,B 0.000,C 90.000,E1 67.358} C_DIS
LIN {X 0.009,Y -572.879,Z 823.167,A 0.000,B 0.000,C 90.000,E1 65.973} C_DIS
LIN {X 0.240,Y -572.306,Z 823.159,A 0.000,B 0.000,C 90.000,E1 64.588} C_DIS
LIN {X -0.062,Y -571.615,Z 823.151,A 0.000,B 0.000,C 90.000,E1 63.256} C_DIS
LIN {X -0.121,Y -570.768,Z 823.144,A 0.000,B 0.000,C 90.000,E1 61.897} C_DIS
LIN {X -0.201,Y -569.586,Z 823.136,A 0.000,B 0.000,C 90.000,E1 60.539} C_DIS
LIN {X 0.151,Y -568.365,Z 823.130,A 0.000,B 0.000,C 90.000,E1 59.410} C_DIS
LIN {X -0.189,Y -566.697,Z 823.123,A 0.000,B 0.000,C 90.000,E1 58.074} C_DIS
LIN {X -0.057,Y -565.032,Z 823.116,A 0.000,B 0.000,C 90.000,E1 56.962} C_DIS
LIN {X -0.045,Y -563.665,Z 823.112,A 0.000,B 0.000,C 90.000,E1 56.135} C_DIS
LIN {X -0.048,Y -562.130,Z 823.107,A 0.000,B 0.000,C 90.000,E1 55.308} C_DIS
LIN {X -0.071,Y -560.397,Z 823.103,A 0.000,B 0.000,C 90.000,E1 54.482} C_DIS
LIN {X 0.301,Y -557.838,Z 823.097,A 0.000,B 0.000,C 90.000,E1 53.336} C_DIS
LIN {X -0.223,Y -555.647,Z 823.092,A 0.000,B 0.000,C 90.000,E1 52.557} C_DIS
LIN {X 0.005,Y -553.195,Z 823.087,A 0.000,B 0.000,C 90.000,E1 51.698} C_DIS
LIN {X -0.229,Y -550.464,Z 823.083,A 0.000,B 0.000,C 90.000,E1 50.884} C_DIS
LIN {X -0.090,Y -546.196,Z 823.076,A 0.000,B 0.000,C 90.000,E1 49.747} C_DIS
LIN {X 0.148,Y -544.494,Z 823.074,A 0.000,B 0.000,C 90.000,E1 49.299} C_DIS
LIN {X -0.011,Y -541.318,Z 823.070,A 0.000,B 0.000,C 90.000,E1 48.609} C_DIS
LIN {X 0.018,Y -538.608,Z 823.067,A 0.000,B 0.000,C 90.000,E1 48.038} C_DIS
LIN {X -0.015,Y -535.643,Z 823.064,A 0.000,B 0.000,C 90.000,E1 47.472} C_DIS
LIN {X 0.107,Y -531.458,Z 823.060,A 0.000,B 0.000,C 90.000,E1 46.743} C_DIS
LIN {X -0.334,Y -527.761,Z 823.057,A 0.000,B 0.000,C 90.000,E1 46.215} C_DIS
LIN {X 0.306,Y -523.736,Z 823.053,A 0.000,B 0.000,C 90.000,E1 45.567} C_DIS
LIN {X 0.174,Y -519.404,Z 823.050,A 0.000,B 0.000,C 90.000,E1 45.000} C_DIS
LIN {X -0.125,Y -515.900,Z 823.048,A 0.000,B 0.000,C 90.000,E1 44.595} C_DIS
LIN {X -0.161,Y -509.456,Z 823.044,A 0.000,B 0.000,C 90.000,E1 43.866} C_DIS
LIN {X -0.066,Y -505.474,Z 823.041,A 0.000,B 0.000,C 90.000,E1 43.419} C_DIS
LIN {X -0.212,Y -501.349,Z 823.039,A 0.000,B 0.000,C 90.000,E1 43.014} C_DIS
LIN {X -0.011,Y -495.590,Z 823.036,A 0.000,B 0.000,C 90.000,E1 42.447} C_DIS
LIN {X -0.038,Y -491.677,Z 823.034,A 0.000,B 0.000,C 90.000,E1 42.081} C_DIS
LIN {X 0.105,Y -485.717,Z 823.031,A 0.000,B 0.000,C 90.000,E1 41.553} C_DIS
LIN {X 0.059,Y -478.016,Z 823.028,A 0.000,B 0.000,C 90.000,E1 40.943} C_DIS
LIN {X 0.097,Y -470.188,Z 823.024,A 0.000,B 0.000,C 90.000,E1 40.334} C_DIS
LIN {X 0.098,Y -457.435,Z 823.019,A 0.000,B 0.000,C 90.000,E1 39.402} C_DIS
LIN {X 0.069,Y -443.370,Z 823.013,A 0.000,B 0.000,C 90.000,E1 38.382} C_DIS
LIN {X -0.014,Y -418.450,Z 823.003,A 0.000,B 0.000,C 90.000,E1 36.457} C_DIS
LIN {X 0.038,Y -406.448,Z 822.997,A 0.000,B 0.000,C 90.000,E1 35.391} C_DIS
LIN {X 0.245,Y -401.063,Z 822.994,A 0.000,B 0.000,C 90.000,E1 34.818} C_DIS
LIN {X 0.114,Y -399.795,Z 822.993,A 0.000,B 0.000,C 90.000,E1 34.692} C_DIS
LIN {X -0.170,Y -397.698,Z 822.991,A 0.000,B 0.000,C 90.000,E1 34.405} C_DIS
LIN {X -0.207,Y -397.679,Z 822.991,A 0.000,B 0.000,C 90.000,E1 34.405} C_DIS
LIN {X -0.211,Y -393.988,Z 822.978,A 0.000,B 0.000,C 90.000,E1 32.005} C_DIS
LIN {X -0.012,Y -392.244,Z 822.972,A 0.000,B 0.000,C 90.000,E1 31.003} C_DIS
LIN {X 0.013,Y -393.734,Z 822.954,A 0.000,B 0.000,C 90.000,E1 27.719} C_DIS
LIN {X -0.063,Y -395.536,Z 822.938,A 0.000,B 0.000,C 90.000,E1 24.899} C_DIS
LIN {X 0.024,Y -397.088,Z 822.927,A 0.000,B 0.000,C 90.000,E1 22.770} C_DIS
LIN {X 0.143,Y -399.389,Z 822.911,A 0.000,B 0.000,C 90.000,E1 19.939} C_DIS
LIN {X 0.032,Y -402.771,Z 822.893,A 0.000,B 0.000,C 90.000,E1 16.804} C_DIS
LIN {X -0.178,Y -408.051,Z 822.872,A 0.000,B 0.000,C 90.000,E1 13.008} C_DIS
LIN {X 0.116,Y -411.405,Z 822.861,A 0.000,B 0.000,C 90.000,E1 10.894} C_DIS
LIN {X -0.025,Y -415.582,Z 822.847,A 0.000,B 0.000,C 90.000,E1 8.511} C_DIS
LIN {X -0.180,Y -419.295,Z 822.836,A 0.000,B 0.000,C 90.000,E1 6.486} C_DIS
LIN {X 0.114,Y -423.628,Z 822.823,A 0.000,B 0.000,C 90.000,E1 4.073} C_DIS
LIN {X 0.111,Y -428.273,Z 822.810,A 0.000,B 0.000,C 90.000,E1 1.718} C_DIS
LIN {X -0.015,Y -434.665,Z 822.793,A 0.000,B 0.000,C 90.000,E1 358.797} C_DIS
LIN {X -0.057,Y -440.904,Z 822.779,A 0.000,B 0.000,C 90.000,E1 356.159} C_DIS
LIN {X -0.136,Y -445.745,Z 822.768,A 0.000,B 0.000,C 90.000,E1 354.204} C_DIS
LIN {X 0.099,Y -453.536,Z 822.752,A 0.000,B 0.000,C 90.000,E1 351.254} C_DIS
LIN {X -0.002,Y -455.964,Z 822.748,A 0.000,B 0.000,C 90.000,E1 350.622} C_DIS
LIN {X -0.041,Y -457.182,Z 822.747,A 0.000,B 0.000,C 90.000,E1 350.387} C_DIS
LIN {X 0.120,Y -458.946,Z 822.745,A 0.000,B 0.000,C 90.000,E1 350.095} C_DIS
LIN {X -0.193,Y -461.000,Z 822.744,A 0.000,B 0.000,C 90.000,E1 349.859} C_DIS
LIN {X -0.116,Y -462.467,Z 822.743,A 0.000,B 0.000,C 90.000,E1 349.690} C_DIS
LIN {X -0.017,Y -467.966,Z 822.740,A 0.000,B 0.000,C 90.000,E1 349.218} C_DIS
LIN {X -0.107,Y -473.871,Z 822.738,A 0.000,B 0.000,C 90.000,E1 348.814} C_DIS
LIN {X -0.245,Y -487.919,Z 822.733,A 0.000,B 0.000,C 90.000,E1 347.937} C_DIS
LIN {X -0.029,Y -502.157,Z 822.728,A 0.000,B 0.000,C 90.000,E1 346.992} C_DIS
LIN {X 0.236,Y -513.134,Z 822.724,A 0.000,B 0.000,C 90.000,E1 346.228} C_DIS
LIN {X -0.157,Y -525.534,Z 822.719,A 0.000,B 0.000,C 90.000,E1 345.408} C_DIS
LIN {X -0.105,Y -536.162,Z 822.715,A 0.000,B 0.000,C 90.000,E1 344.629} C_DIS
LIN {X 0.131,Y -544.919,Z 822.711,A 0.000,B 0.000,C 90.000,E1 343.921} C_DIS
LIN {X -0.141,Y -551.848,Z 822.708,A 0.000,B 0.000,C 90.000,E1 343.378} C_DIS
LIN {X -0.261,Y -558.748,Z 822.704,A 0.000,B 0.000,C 90.000,E1 342.779} C_DIS
LIN {X 0.119,Y -564.016,Z 822.701,A 0.000,B 0.000,C 90.000,E1 342.236} C_DIS
LIN {X 0.104,Y -570.370,Z 822.698,A 0.000,B 0.000,C 90.000,E1 341.583} C_DIS
LIN {X 0.084,Y -576.514,Z 822.694,A 0.000,B 0.000,C 90.000,E1 340.913} C_DIS
LIN {X 0.184,Y -579.967,Z 822.692,A 0.000,B 0.000,C 90.000,E1 340.496} C_DIS
LIN {X 0.146,Y -585.262,Z 822.688,A 0.000,B 0.000,C 90.000,E1 339.826} C_DIS
LIN {X 0.152,Y -590.132,Z 822.684,A 0.000,B 0.000,C 90.000,E1 339.156} C_DIS
LIN {X -0.136,Y -594.592,Z 822.681,A 0.000,B 0.000,C 90.000,E1 338.518} C_DIS
LIN {X -0.135,Y -600.269,Z 822.675,A 0.000,B 0.000,C 90.000,E1 337.592} C_DIS
LIN {X -0.068,Y -605.792,Z 822.670,A 0.000,B 0.000,C 90.000,E1 336.666} C_DIS
LIN {X 0.058,Y -611.142,Z 822.665,A 0.000,B 0.000,C 90.000,E1 335.741} C_DIS
LIN {X -0.071,Y -616.994,Z 822.660,A 0.000,B 0.000,C 90.000,E1 334.717} C_DIS
LIN {X -0.114,Y -622.398,Z 822.654,A 0.000,B 0.000,C 90.000,E1 333.691} C_DIS
LIN {X -0.084,Y -627.480,Z 822.648,A 0.000,B 0.000,C 90.000,E1 332.666} C_DIS
LIN {X -0.023,Y -630.996,Z 822.644,A 0.000,B 0.000,C 90.000,E1 331.897} C_DIS
LIN {X 0.102,Y -635.592,Z 822.638,A 0.000,B 0.000,C 90.000,E1 330.873} C_DIS
LIN {X 0.040,Y -640.060,Z 822.633,A 0.000,B 0.000,C 90.000,E1 329.871} C_DIS
LIN {X -0.406,Y -642.193,Z 822.630,A 0.000,B 0.000,C 90.000,E1 329.410} C_DIS
LIN {X -0.042,Y -646.132,Z 822.624,A 0.000,B 0.000,C 90.000,E1 328.377} C_DIS
LIN {X 0.044,Y -649.833,Z 822.619,A 0.000,B 0.000,C 90.000,E1 327.375} C_DIS
LIN {X 0.088,Y -652.380,Z 822.615,A 0.000,B 0.000,C 90.000,E1 326.628} C_DIS
LIN {X -0.303,Y -657.173,Z 822.606,A 0.000,B 0.000,C 90.000,E1 325.182} C_DIS
LIN {X 0.212,Y -660.673,Z 822.600,A 0.000,B 0.000,C 90.000,E1 323.909} C_DIS
LIN {X 0.296,Y -663.280,Z 822.594,A 0.000,B 0.000,C 90.000,E1 322.924} C_DIS
LIN {X -0.145,Y -666.206,Z 822.587,A 0.000,B 0.000,C 90.000,E1 321.743} C_DIS
LIN {X -0.092,Y -667.775,Z 822.583,A 0.000,B 0.000,C 90.000,E1 321.009} C_DIS
LIN {X 0.053,Y -670.267,Z 822.577,A 0.000,B 0.000,C 90.000,E1 319.784} C_DIS
LIN {X 0.151,Y -672.514,Z 822.570,A 0.000,B 0.000,C 90.000,E1 318.566} C_DIS
LIN {X -0.236,Y -674.276,Z 822.565,A 0.000,B 0.000,C 90.000,E1 317.634} C_DIS
LIN {X -0.165,Y -675.449,Z 822.561,A 0.000,B 0.000,C 90.000,E1 316.905} C_DIS
LIN {X 0.037,Y -677.476,Z 822.553,A 0.000,B 0.000,C 90.000,E1 315.445} C_DIS
LIN {X -0.374,Y -678.153,Z 822.550,A 0.000,B 0.000,C 90.000,E1 315.000} C_DIS
LIN {X -0.136,Y -679.845,Z 822.542,A 0.000,B 0.000,C 90.000,E1 313.542} C_DIS
LIN {X 0.162,Y -681.505,Z 822.534,A 0.000,B 0.000,C 90.000,E1 312.081} C_DIS
LIN {X -0.020,Y -683.100,Z 822.526,A 0.000,B 0.000,C 90.000,E1 310.663} C_DIS
LIN {X -0.159,Y -684.302,Z 822.519,A 0.000,B 0.000,C 90.000,E1 309.483} C_DIS
LIN {X 0.305,Y -685.598,Z 822.511,A 0.000,B 0.000,C 90.000,E1 308.016} C_DIS
LIN {X 0.375,Y -686.857,Z 822.503,A 0.000,B 0.000,C 90.000,E1 306.583} C_DIS
LIN {X -0.123,Y -687.807,Z 822.497,A 0.000,B 0.000,C 90.000,E1 305.438} C_DIS
LIN {X -0.052,Y -688.686,Z 822.490,A 0.000,B 0.000,C 90.000,E1 304.246} C_DIS
LIN {X -0.139,Y -689.674,Z 822.482,A 0.000,B 0.000,C 90.000,E1 302.832} C_DIS
LIN {X -0.418,Y -690.561,Z 822.476,A 0.000,B 0.000,C 90.000,E1 301.671} C_DIS
LIN {X -0.099,Y -691.424,Z 822.469,A 0.000,B 0.000,C 90.000,E1 300.463} C_DIS
LIN {X 0.126,Y -692.438,Z 822.461,A 0.000,B 0.000,C 90.000,E1 299.027} C_DIS
LIN {X 0.010,Y -693.627,Z 822.452,A 0.000,B 0.000,C 90.000,E1 297.385} C_DIS
LIN {X 0.208,Y -694.962,Z 822.443,A 0.000,B 0.000,C 90.000,E1 295.720} C_DIS
LIN {X -0.120,Y -696.095,Z 822.435,A 0.000,B 0.000,C 90.000,E1 294.335} C_DIS
LIN {X 0.389,Y -696.095,Z 822.433,A 0.000,B 0.000,C 90.000,E1 293.823} C_DIS
LIN {X -0.276,Y -695.934,Z 822.431,A 0.000,B 0.000,C 90.000,E1 293.643} C_DIS
LIN {X -0.045,Y -694.914,Z 822.429,A 0.000,B 0.000,C 90.000,E1 293.153} C_DIS
LIN {X 0.204,Y -694.058,Z 822.427,A 0.000,B 0.000,C 90.000,E1 292.898} C_DIS
LIN {X -0.189,Y -692.250,Z 822.426,A 0.000,B 0.000,C 90.000,E1 292.695} C_DIS
LIN {X -0.214,Y -690.273,Z 822.425,A 0.000,B 0.000,C 90.000,E1 292.461} C_DIS
LIN {X -0.099,Y -689.112,Z 822.424,A 0.000,B 0.000,C 90.000,E1 292.333} C_DIS
LIN {X 0.017,Y -687.651,Z 822.423,A 0.000,B 0.000,C 90.000,E1 292.206} C_DIS
LIN {X 0.206,Y -681.894,Z 822.422,A 0.000,B 0.000,C 90.000,E1 291.897} C_DIS
LIN {X -0.033,Y -678.224,Z 822.421,A 0.000,B 0.000,C 90.000,E1 291.770} C_DIS
LIN {X 0.128,Y -672.286,Z 822.420,A 0.000,B 0.000,C 90.000,E1 291.589} C_DIS
LIN {X -0.243,Y -663.604,Z 822.419,A 0.000,B 0.000,C 90.000,E1 291.461} C_DIS
LIN {X -0.111,Y -645.811,Z 822.417,A 0.000,B 0.000,C 90.000,E1 291.153} C_DIS
LIN {X 0.222,Y -635.242,Z 822.416,A 0.000,B 0.000,C 90.000,E1 290.918} C_DIS
LIN {X -0.350,Y -626.069,Z 822.415,A 0.000,B 0.000,C 90.000,E1 290.737} C_DIS
LIN {X 0.060,Y -623.435,Z 822.415,A 0.000,B 0.000,C 90.000,E1 290.610} C_DIS
LIN {X 0.018,Y -621.349,Z 822.414,A 0.000,B 0.000,C 90.000,E1 290.556} C_DIS
LIN {X 0.090,Y -618.190,Z 822.414,A 0.000,B 0.000,C 90.000,E1 290.429} C_DIS
LIN {X -0.140,Y -615.306,Z 822.413,A 0.000,B 0.000,C 90.000,E1 290.301} C_DIS
LIN {X 0.152,Y -611.949,Z 822.412,A 0.000,B 0.000,C 90.000,E1 290.120} C_DIS
LIN {X 0.056,Y -609.828,Z 822.411,A 0.000,B 0.000,C 90.000,E1 289.939} C_DIS
LIN {X 0.016,Y -609.807,Z 822.411,A 0.000,B 0.000,C 90.000,E1 289.939} C_DIS
LIN {X -0.232,Y -609.258,Z 822.410,A 0.000,B 0.000,C 90.000,E1 289.758} C_DIS
LIN {X 0.282,Y -609.929,Z 822.408,A 0.000,B 0.000,C 90.000,E1 289.450} C_DIS
LIN {X 0.204,Y -610.860,Z 822.407,A 0.000,B 0.000,C 90.000,E1 289.214} C_DIS
LIN {X 0.195,Y -618.398,Z 822.400,A 0.000,B 0.000,C 90.000,E1 287.946} C_DIS
LIN {X -0.082,Y -621.095,Z 822.397,A 0.000,B 0.000,C 90.000,E1 287.457} C_DIS
LIN {X 0.251,Y -623.393,Z 822.394,A 0.000,B 0.000,C 90.000,E1 286.913} C_DIS
LIN {X -0.184,Y -625.503,Z 822.391,A 0.000,B 0.000,C 90.000,E1 286.441} C_DIS
LIN {X -0.032,Y -628.079,Z 822.387,A 0.000,B 0.000,C 90.000,E1 285.662} C_DIS
LIN {X 0.175,Y -629.539,Z 822.384,A 0.000,B 0.000,C 90.000,E1 285.134} C_DIS
LIN {X -0.246,Y -631.233,Z 822.380,A 0.000,B 0.000,C 90.000,E1 284.411} C_DIS
LIN {X -0.015,Y -632.079,Z 822.377,A 0.000,B 0.000,C 90.000,E1 283.883} C_DIS
LIN {X 0.041,Y -632.784,Z 822.373,A 0.000,B 0.000,C 90.000,E1 283.119} C_DIS
LIN {X 0.289,Y -633.016,Z 822.370,A 0.000,B 0.000,C 90.000,E1 282.591} C_DIS
LIN {X -0.079,Y -632.786,Z 822.367,A 0.000,B 0.000,C 90.000,E1 282.119} C_DIS
LIN {X -0.145,Y -631.706,Z 822.363,A 0.000,B 0.000,C 90.000,E1 281.366} C_DIS
LIN {X 0.097,Y -630.707,Z 822.360,A 0.000,B 0.000,C 90.000,E1 280.838} C_DIS
LIN {X 0.330,Y -629.366,Z 822.357,A 0.000,B 0.000,C 90.000,E1 280.310} C_DIS
LIN {X -0.178,Y -627.735,Z 822.355,A 0.000,B 0.000,C 90.000,E1 279.849} C_DIS
LIN {X -0.125,Y -625.065,Z 822.351,A 0.000,B 0.000,C 90.000,E1 279.208} C_DIS
LIN {X 0.058,Y -622.366,Z 822.348,A 0.000,B 0.000,C 90.000,E1 278.681} C_DIS
LIN {X 0.125,Y -619.222,Z 822.345,A 0.000,B 0.000,C 90.000,E1 278.163} C_DIS
LIN {X 0.173,Y -615.435,Z 822.343,A 0.000,B 0.000,C 90.000,E1 277.644} C_DIS
LIN {X -0.075,Y -613.113,Z 822.341,A 0.000,B 0.000,C 90.000,E1 277.409} C_DIS
LIN {X 0.134,Y -609.481,Z 822.339,A 0.000,B 0.000,C 90.000,E1 277.004} C_DIS
LIN {X -0.036,Y -608.000,Z 822.338,A 0.000,B 0.000,C 90.000,E1 276.891} C_DIS
LIN {X 0.013,Y -601.941,Z 822.336,A 0.000,B 0.000,C 90.000,E1 276.429} C_DIS
LIN {X -0.127,Y -593.668,Z 822.333,A 0.000,B 0.000,C 90.000,E1 275.967} C_DIS
LIN {X -0.090,Y -584.506,Z 822.331,A 0.000,B 0.000,C 90.000,E1 275.568} C_DIS
LIN {X 0.257,Y -581.107,Z 822.330,A 0.000,B 0.000,C 90.000,E1 275.391} C_DIS
LIN {X 0.095,Y -573.302,Z 822.329,A 0.000,B 0.000,C 90.000,E1 275.163} C_DIS
LIN {X 0.011,Y -566.822,Z 822.328,A 0.000,B 0.000,C 90.000,E1 275.049} C_DIS
LIN {X -0.205,Y -560.201,Z 822.328,A 0.000,B 0.000,C 90.000,E1 275.049} C_DIS
LIN {X -0.239,Y -552.372,Z 822.328,A 0.000,B 0.000,C 90.000,E1 275.049} C_DIS
LIN {X -0.274,Y -552.136,Z 822.328,A 0.000,B 0.000,C 90.000,E1 275.049} C_DIS
LIN {X 0.229,Y -552.090,Z 822.328,A 0.000,B 0.000,C 90.000,E1 274.992} C_DIS
LIN {X 0.197,Y -551.213,Z 822.327,A 0.000,B 0.000,C 90.000,E1 274.821} C_DIS
LIN {X -0.170,Y -549.793,Z 822.326,A 0.000,B 0.000,C 90.000,E1 274.645} C_DIS
LIN {X -0.212,Y -549.766,Z 822.326,A 0.000,B 0.000,C 90.000,E1 274.645} C_DIS
LIN {X 0.228,Y -548.708,Z 822.320,A 0.000,B 0.000,C 90.000,E1 273.555} C_DIS
LIN {X -0.054,Y -547.705,Z 822.312,A 0.000,B 0.000,C 90.000,E1 272.178} C_DIS
LIN {X 0.236,Y -546.516,Z 822.303,A 0.000,B 0.000,C 90.000,E1 270.458} C_DIS
LIN {X -0.021,Y -545.121,Z 822.292,A 0.000,B 0.000,C 90.000,E1 268.511} C_DIS
LIN {X -0.251,Y -543.586,Z 822.279,A 0.000,B 0.000,C 90.000,E1 266.274} C_DIS
LIN {X -0.068,Y -542.885,Z 822.273,A 0.000,B 0.000,C 90.000,E1 265.122} C_DIS
LIN {X 0.122,Y -541.940,Z 822.265,A 0.000,B 0.000,C 90.000,E1 263.685} C_DIS
LIN {X -0.191,Y -540.735,Z 822.257,A 0.000,B 0.000,C 90.000,E1 262.299} C_DIS
LIN {X 0.160,Y -539.177,Z 822.248,A 0.000,B 0.000,C 90.000,E1 260.557} C_DIS
LIN {X -0.120,Y -537.775,Z 822.240,A 0.000,B 0.000,C 90.000,E1 259.162} C_DIS
LIN {X 0.199,Y -536.338,Z 822.232,A 0.000,B 0.000,C 90.000,E1 257.701} C_DIS
LIN {X -0.093,Y -535.235,Z 822.225,A 0.000,B 0.000,C 90.000,E1 256.589} C_DIS
LIN {X -0.048,Y -533.273,Z 822.216,A 0.000,B 0.000,C 90.000,E1 254.866} C_DIS
LIN {X -0.014,Y -530.999,Z 822.205,A 0.000,B 0.000,C 90.000,E1 252.851} C_DIS
LIN {X 0.053,Y -529.574,Z 822.198,A 0.000,B 0.000,C 90.000,E1 251.692} C_DIS
LIN {X 0.115,Y -527.745,Z 822.190,A 0.000,B 0.000,C 90.000,E1 250.242} C_DIS
LIN {X -0.172,Y -525.755,Z 822.182,A 0.000,B 0.000,C 90.000,E1 248.827} C_DIS
LIN {X 0.156,Y -523.280,Z 822.173,A 0.000,B 0.000,C 90.000,E1 247.050} C_DIS
LIN {X 0.131,Y -520.587,Z 822.163,A 0.000,B 0.000,C 90.000,E1 245.305} C_DIS
LIN {X 0.121,Y -518.204,Z 822.155,A 0.000,B 0.000,C 90.000,E1 243.845} C_DIS
LIN {X -0.059,Y -516.230,Z 822.148,A 0.000,B 0.000,C 90.000,E1 242.692} C_DIS
LIN {X -0.026,Y -514.105,Z 822.142,A 0.000,B 0.000,C 90.000,E1 241.513} C_DIS
LIN {X -0.031,Y -510.859,Z 822.132,A 0.000,B 0.000,C 90.000,E1 239.744} C_DIS
LIN {X -0.153,Y -509.256,Z 822.127,A 0.000,B 0.000,C 90.000,E1 238.869} C_DIS
LIN {X 0.037,Y -506.904,Z 822.120,A 0.000,B 0.000,C 90.000,E1 237.661} C_DIS
LIN {X 0.148,Y -505.056,Z 822.115,A 0.000,B 0.000,C 90.000,E1 236.755} C_DIS
LIN {X 0.148,Y -501.812,Z 822.107,A 0.000,B 0.000,C 90.000,E1 235.261} C_DIS
LIN {X -0.175,Y -497.668,Z 822.097,A 0.000,B 0.000,C 90.000,E1 233.497} C_DIS
LIN {X 0.015,Y -493.287,Z 822.087,A 0.000,B 0.000,C 90.000,E1 231.662} C_DIS
LIN {X 0.112,Y -490.326,Z 822.080,A 0.000,B 0.000,C 90.000,E1 230.436} C_DIS
LIN {X -0.101,Y -485.394,Z 822.068,A 0.000,B 0.000,C 90.000,E1 228.324} C_DIS
LIN {X 0.072,Y -481.176,Z 822.058,A 0.000,B 0.000,C 90.000,E1 226.458} C_DIS
LIN {X 0.250,Y -476.521,Z 822.046,A 0.000,B 0.000,C 90.000,E1 224.271} C_DIS
LIN {X -0.260,Y -471.136,Z 822.032,A 0.000,B 0.000,C 90.000,E1 221.838} C_DIS
LIN {X -0.059,Y -467.164,Z 822.022,A 0.000,B 0.000,C 90.000,E1 219.930} C_DIS
LIN {X 0.059,Y -463.885,Z 822.013,A 0.000,B 0.000,C 90.000,E1 218.338} C_DIS
LIN {X -0.116,Y -459.283,Z 822.001,A 0.000,B 0.000,C 90.000,E1 216.137} C_DIS
LIN {X -0.054,Y -455.991,Z 821.992,A 0.000,B 0.000,C 90.000,E1 214.532} C_DIS
LIN {X -0.027,Y -450.601,Z 821.978,A 0.000,B 0.000,C 90.000,E1 211.957} C_DIS
LIN {X 0.077,Y -446.579,Z 821.967,A 0.000,B 0.000,C 90.000,E1 210.001} C_DIS
LIN {X 0.182,Y -443.395,Z 821.958,A 0.000,B 0.000,C 90.000,E1 208.359} C_DIS
LIN {X 0.051,Y -439.528,Z 821.947,A 0.000,B 0.000,C 90.000,E1 206.411} C_DIS
LIN {X 0.173,Y -436.914,Z 821.940,A 0.000,B 0.000,C 90.000,E1 205.079} C_DIS
LIN {X -0.097,Y -433.569,Z 821.930,A 0.000,B 0.000,C 90.000,E1 203.462} C_DIS
LIN {X -0.050,Y -429.696,Z 821.919,A 0.000,B 0.000,C 90.000,E1 201.461} C_DIS
LIN {X -0.016,Y -425.874,Z 821.908,A 0.000,B 0.000,C 90.000,E1 199.450} C_DIS
LIN {X -0.209,Y -421.877,Z 821.897,A 0.000,B 0.000,C 90.000,E1 197.457} C_DIS
LIN {X 0.184,Y -417.950,Z 821.886,A 0.000,B 0.000,C 90.000,E1 195.371} C_DIS
LIN {X -0.073,Y -414.760,Z 821.876,A 0.000,B 0.000,C 90.000,E1 193.703} C_DIS
LIN {X -0.187,Y -411.506,Z 821.867,A 0.000,B 0.000,C 90.000,E1 192.007} C_DIS
LIN {X 0.042,Y -408.198,Z 821.857,A 0.000,B 0.000,C 90.000,E1 190.254} C_DIS
LIN {X 0.128,Y -404.946,Z 821.847,A 0.000,B 0.000,C 90.000,E1 188.511} C_DIS
LIN {X 0.082,Y -401.080,Z 821.836,A 0.000,B 0.000,C 90.000,E1 186.429} C_DIS
LIN {X -0.084,Y -394.087,Z 821.812,A 0.000,B 0.000,C 90.000,E1 182.236} C_DIS
LIN {X -0.144,Y -388.932,Z 821.791,A 0.000,B 0.000,C 90.000,E1 178.339} C_DIS
LIN {X -0.112,Y -387.214,Z 821.783,A 0.000,B 0.000,C 90.000,E1 176.906} C_DIS
LIN {X 0.110,Y -384.695,Z 821.771,A 0.000,B 0.000,C 90.000,E1 174.723} C_DIS
LIN {X -0.160,Y -381.861,Z 821.757,A 0.000,B 0.000,C 90.000,E1 172.243} C_DIS
LIN {X 0.159,Y -380.125,Z 821.747,A 0.000,B 0.000,C 90.000,E1 170.387} C_DIS
LIN {X 0.136,Y -378.491,Z 821.737,A 0.000,B 0.000,C 90.000,E1 168.578} C_DIS
LIN {X -0.084,Y -376.030,Z 821.721,A 0.000,B 0.000,C 90.000,E1 165.700} C_DIS
LIN {X 0.079,Y -373.389,Z 821.690,A 0.000,B 0.000,C 90.000,E1 160.188} C_DIS
LIN {X 0.060,Y -373.365,Z 821.680,A 0.000,B 0.000,C 90.000,E1 158.358} C_DIS
LIN {X -0.023,Y -373.912,Z 821.670,A 0.000,B 0.000,C 90.000,E1 156.538} C_DIS
LIN {X 0.056,Y -374.408,Z 821.666,A 0.000,B 0.000,C 90.000,E1 155.793} C_DIS
LIN {X 0.004,Y -376.347,Z 821.655,A 0.000,B 0.000,C 90.000,E1 153.973} C_DIS
LIN {X -0.079,Y -377.385,Z 821.651,A 0.000,B 0.000,C 90.000,E1 153.256} C_DIS
LIN {X 0.187,Y -378.786,Z 821.647,A 0.000,B 0.000,C 90.000,E1 152.487} C_DIS
LIN {X 0.127,Y -380.468,Z 821.643,A 0.000,B 0.000,C 90.000,E1 151.769} C_DIS
LIN {X -0.022,Y -384.218,Z 821.636,A 0.000,B 0.000,C 90.000,E1 150.539} C_DIS
LIN {X 0.149,Y -384.852,Z 821.635,A 0.000,B 0.000,C 90.000,E1 150.333} C_DIS
LIN {X 0.018,Y -388.705,Z 821.631,A 0.000,B 0.000,C 90.000,E1 149.537} C_DIS
LIN {X 0.203,Y -389.528,Z 821.630,A 0.000,B 0.000,C 90.000,E1 149.331} C_DIS
LIN {X 0.002,Y -392.036,Z 821.627,A 0.000,B 0.000,C 90.000,E1 148.918} C_DIS
LIN {X 0.195,Y -395.081,Z 821.625,A 0.000,B 0.000,C 90.000,E1 148.456} C_DIS
LIN {X -0.202,Y -397.688,Z 821.623,A 0.000,B 0.000,C 90.000,E1 148.201} C_DIS
LIN {X 0.193,Y -403.009,Z 821.620,A 0.000,B 0.000,C 90.000,E1 147.582} C_DIS
LIN {X -0.229,Y -411.891,Z 821.616,A 0.000,B 0.000,C 90.000,E1 146.914} C_DIS
LIN {X -0.128,Y -423.976,Z 821.612,A 0.000,B 0.000,C 90.000,E1 146.087} C_DIS
LIN {X -0.025,Y -432.657,Z 821.609,A 0.000,B 0.000,C 90.000,E1 145.548} C_DIS
LIN {X -0.001,Y -440.029,Z 821.606,A 0.000,B 0.000,C 90.000,E1 145.022} C_DIS
LIN {X -0.199,Y -450.971,Z 821.601,A 0.000,B 0.000,C 90.000,E1 144.196} C_DIS
LIN {X 0.225,Y -456.553,Z 821.598,A 0.000,B 0.000,C 90.000,E1 143.623} C_DIS
LIN {X -0.124,Y -465.967,Z 821.592,A 0.000,B 0.000,C 90.000,E1 142.637} C_DIS
LIN {X -0.039,Y -474.865,Z 821.586,A 0.000,B 0.000,C 90.000,E1 141.537} C_DIS
LIN {X 0.208,Y -479.168,Z 821.583,A 0.000,B 0.000,C 90.000,E1 140.884} C_DIS
LIN {X 0.139,Y -483.804,Z 821.579,A 0.000,B 0.000,C 90.000,E1 140.275} C_DIS
LIN {X 0.087,Y -488.139,Z 821.576,A 0.000,B 0.000,C 90.000,E1 139.666} C_DIS
LIN {X -0.092,Y -494.199,Z 821.571,A 0.000,B 0.000,C 90.000,E1 138.771} C_DIS
LIN {X 0.085,Y -501.965,Z 821.563,A 0.000,B 0.000,C 90.000,E1 137.391} C_DIS
LIN {X -0.092,Y -506.099,Z 821.559,A 0.000,B 0.000,C 90.000,E1 136.662} C_DIS
LIN {X 0.261,Y -510.926,Z 821.554,A 0.000,B 0.000,C 90.000,E1 135.729} C_DIS
LIN {X 0.171,Y -514.557,Z 821.550,A 0.000,B 0.000,C 90.000,E1 135.000} C_DIS
LIN {X -0.024,Y -517.641,Z 821.547,A 0.000,B 0.000,C 90.000,E1 134.433} C_DIS
LIN {X 0.087,Y -521.995,Z 821.542,A 0.000,B 0.000,C 90.000,E1 133.542} C_DIS
LIN {X 0.172,Y -524.240,Z 821.540,A 0.000,B 0.000,C 90.000,E1 133.095} C_DIS
LIN {X 0.197,Y -527.595,Z 821.536,A 0.000,B 0.000,C 90.000,E1 132.366} C_DIS
LIN {X -0.132,Y -532.032,Z 821.530,A 0.000,B 0.000,C 90.000,E1 131.391} C_DIS
LIN {X 0.106,Y -537.704,Z 821.522,A 0.000,B 0.000,C 90.000,E1 129.930} C_DIS
LIN {X -0.272,Y -541.669,Z 821.516,A 0.000,B 0.000,C 90.000,E1 128.830} C_DIS
LIN {X 0.137,Y -544.286,Z 821.511,A 0.000,B 0.000,C 90.000,E1 127.935} C_DIS
LIN {X 0.000,Y -548.366,Z 821.503,A 0.000,B 0.000,C 90.000,E1 126.537} C_DIS
LIN {X 0.100,Y -549.649,Z 821.500,A 0.000,B 0.000,C 90.000,E1 125.964} C_DIS
LIN {X 0.209,Y -550.631,Z 821.497,A 0.000,B 0.000,C 90.000,E1 125.391} C_DIS
LIN {X 0.323,Y -551.414,Z 821.494,A 0.000,B 0.000,C 90.000,E1 124.818} C_DIS
LIN {X 0.188,Y -552.199,Z 821.489,A 0.000,B 0.000,C 90.000,E1 123.992} C_DIS
LIN {X 0.062,Y -552.348,Z 821.484,A 0.000,B 0.000,C 90.000,E1 123.166} C_DIS
LIN {X -0.065,Y -552.765,Z 821.480,A 0.000,B 0.000,C 90.000,E1 122.339} C_DIS
LIN {X 0.100,Y -553.217,Z 821.472,A 0.000,B 0.000,C 90.000,E1 120.924} C_DIS
LIN {X -0.081,Y -553.392,Z 821.469,A 0.000,B 0.000,C 90.000,E1 120.384} C_DIS
LIN {X -0.010,Y -553.735,Z 821.464,A 0.000,B 0.000,C 90.000,E1 119.539} C_DIS
LIN {X -0.078,Y -553.852,Z 821.462,A 0.000,B 0.000,C 90.000,E1 119.127} C_DIS
LIN {X -0.024,Y -554.521,Z 821.460,A 0.000,B 0.000,C 90.000,E1 118.821} C_DIS
LIN {X -0.246,Y -554.564,Z 821.459,A 0.000,B 0.000,C 90.000,E1 118.565} C_DIS
LIN {X -0.111,Y -554.232,Z 821.458,A 0.000,B 0.000,C 90.000,E1 118.359} C_DIS
LIN {X 0.285,Y -554.686,Z 821.457,A 0.000,B 0.000,C 90.000,E1 118.231} C_DIS
LIN {X 0.064,Y -555.316,Z 821.456,A 0.000,B 0.000,C 90.000,E1 117.975} C_DIS
LIN {X -0.008,Y -555.262,Z 821.453,A 0.000,B 0.000,C 90.000,E1 117.564} C_DIS
LIN {X 0.081,Y -556.792,Z 821.448,A 0.000,B 0.000,C 90.000,E1 116.616} C_DIS
LIN {X -0.133,Y -557.122,Z 821.446,A 0.000,B 0.000,C 90.000,E1 116.360} C_DIS
LIN {X 0.155,Y -557.043,Z 821.445,A 0.000,B 0.000,C 90.000,E1 116.052} C_DIS
LIN {X -0.056,Y -557.478,Z 821.443,A 0.000,B 0.000,C 90.000,E1 115.796} C_DIS
LIN {X 0.231,Y -559.509,Z 821.433,A 0.000,B 0.000,C 90.000,E1 113.823} C_DIS
LIN {X -0.101,Y -560.372,Z 821.428,A 0.000,B 0.000,C 90.000,E1 113.025} C_DIS
LIN {X -0.206,Y -561.158,Z 821.423,A 0.000,B 0.000,C 90.000,E1 112.206} C_DIS
LIN {X -0.202,Y -562.017,Z 821.417,A 0.000,B 0.000,C 90.000,E1 111.099} C_DIS
LIN {X -0.187,Y -562.531,Z 821.411,A 0.000,B 0.000,C 90.000,E1 109.993} C_DIS
LIN {X 0.175,Y -562.751,Z 821.405,A 0.000,B 0.000,C 90.000,E1 108.852} C_DIS
LIN {X -0.066,Y -562.886,Z 821.396,A 0.000,B 0.000,C 90.000,E1 107.221} C_DIS
LIN {X 0.138,Y -563.553,Z 821.382,A 0.000,B 0.000,C 90.000,E1 104.717} C_DIS
LIN {X -0.245,Y -564.532,Z 821.371,A 0.000,B 0.000,C 90.000,E1 102.827} C_DIS
LIN {X -0.181,Y -565.756,Z 821.360,A 0.000,B 0.000,C 90.000,E1 100.894} C_DIS
LIN {X 0.191,Y -567.006,Z 821.351,A 0.000,B 0.000,C 90.000,E1 99.208} C_DIS
LIN {X -0.058,Y -568.132,Z 821.342,A 0.000,B 0.000,C 90.000,E1 97.587} C_DIS
LIN {X 0.272,Y -569.124,Z 821.333,A 0.000,B 0.000,C 90.000,E1 95.910} C_DIS
LIN {X -0.061,Y -569.909,Z 821.324,A 0.000,B 0.000,C 90.000,E1 94.302} C_DIS
LIN {X 0.065,Y -570.453,Z 821.316,A 0.000,B 0.000,C 90.000,E1 92.922} C_DIS
LIN {X 0.164,Y -570.941,Z 821.309,A 0.000,B 0.000,C 90.000,E1 91.547} C_DIS
LIN {X 0.127,Y -571.315,Z 821.303,A 0.000,B 0.000,C 90.000,E1 90.458} C_DIS
LIN {X -0.069,Y -571.812,Z 821.292,A 0.000,B 0.000,C 90.000,E1 88.568} C_DIS
LIN {X 0.055,Y -572.197,Z 821.284,A 0.000,B 0.000,C 90.000,E1 87.192} C_DIS
LIN {X -0.088,Y -572.569,Z 821.274,A 0.000,B 0.000,C 90.000,E1 85.298} C_DIS
LIN {X 0.266,Y -572.808,Z 821.265,A 0.000,B 0.000,C 90.000,E1 83.628} C_DIS
LIN {X 0.130,Y -573.209,Z 821.256,A 0.000,B 0.000,C 90.000,E1 82.008} C_DIS
LIN {X 0.005,Y -573.652,Z 821.247,A 0.000,B 0.000,C 90.000,E1 80.387} C_DIS
LIN {X -0.024,Y -574.046,Z 821.238,A 0.000,B 0.000,C 90.000,E1 78.757} C_DIS
LIN {X -0.137,Y -574.367,Z 821.230,A 0.000,B 0.000,C 90.000,E1 77.409} C_DIS
LIN {X 0.110,Y -574.481,Z 821.224,A 0.000,B 0.000,C 90.000,E1 76.297} C_DIS
LIN {X -0.072,Y -574.615,Z 821.215,A 0.000,B 0.000,C 90.000,E1 74.685} C_DIS
LIN {X -0.041,Y -574.568,Z 821.207,A 0.000,B 0.000,C 90.000,E1 73.323} C_DIS
LIN {X 0.144,Y -574.491,Z 821.200,A 0.000,B 0.000,C 90.000,E1 71.945} C_DIS
LIN {X 0.135,Y -574.231,Z 821.191,A 0.000,B 0.000,C 90.000,E1 70.315} C_DIS
LIN {X -0.226,Y -573.878,Z 821.182,A 0.000,B 0.000,C 90.000,E1 68.720} C_DIS
LIN {X -0.210,Y -573.465,Z 821.174,A 0.000,B 0.000,C 90.000,E1 67.358} C_DIS
LIN {X -0.135,Y -572.827,Z 821.165,A 0.000,B 0.000,C 90.000,E1 65.717} C_DIS
LIN {X 0.096,Y -572.233,Z 821.158,A 0.000,B 0.000,C 90.000,E1 64.332} C_DIS
LIN {X -0.207,Y -571.482,Z 821.150,A 0.000,B 0.000,C 90.000,E1 62.999} C_DIS
LIN {X -0.101,Y -570.767,Z 821.144,A 0.000,B 0.000,C 90.000,E1 61.897} C_DIS
LIN {X -0.007,Y -569.813,Z 821.138,A 0.000,B 0.000,C 90.000,E1 60.795} C_DIS
LIN {X 0.350,Y -568.651,Z 821.132,A 0.000,B 0.000,C 90.000,E1 59.665} C_DIS
LIN {X -0.090,Y -567.295,Z 821.126,A 0.000,B 0.000,C 90.000,E1 58.614} C_DIS
LIN {X -0.062,Y -566.163,Z 821.121,A 0.000,B 0.000,C 90.000,E1 57.788} C_DIS
LIN {X -0.041,Y -564.918,Z 821.116,A 0.000,B 0.000,C 90.000,E1 56.962} C_DIS
LIN {X -0.030,Y -563.508,Z 821.112,A 0.000,B 0.000,C 90.000,E1 56.135} C_DIS
LIN {X 0.067,Y -561.379,Z 821.106,A 0.000,B 0.000,C 90.000,E1 55.022} C_DIS
LIN {X 0.129,Y -558.891,Z 821.100,A 0.000,B 0.000,C 90.000,E1 53.909} C_DIS
LIN {X 0.060,Y -556.839,Z 821.095,A 0.000,B 0.000,C 90.000,E1 53.084} C_DIS
LIN {X -0.141,Y -554.500,Z 821.090,A 0.000,B 0.000,C 90.000,E1 52.271} C_DIS
LIN {X 0.005,Y -552.837,Z 821.087,A 0.000,B 0.000,C 90.000,E1 51.698} C_DIS
LIN {X -0.231,Y -550.025,Z 821.083,A 0.000,B 0.000,C 90.000,E1 50.884} C_DIS
LIN {X -0.099,Y -545.696,Z 821.076,A 0.000,B 0.000,C 90.000,E1 49.747} C_DIS
LIN {X 0.135,Y -543.945,Z 821.074,A 0.000,B 0.000,C 90.000,E1 49.299} C_DIS
LIN {X -0.029,Y -540.715,Z 821.070,A 0.000,B 0.000,C 90.000,E1 48.609} C_DIS
LIN {X -0.005,Y -537.946,Z 821.067,A 0.000,B 0.000,C 90.000,E1 48.038} C_DIS
LIN {X -0.042,Y -534.919,Z 821.064,A 0.000,B 0.000,C 90.000,E1 47.472} C_DIS
LIN {X -0.097,Y -531.587,Z 821.061,A 0.000,B 0.000,C 90.000,E1 46.905} C_DIS
LIN {X 0.211,Y -527.898,Z 821.057,A 0.000,B 0.000,C 90.000,E1 46.296} C_DIS
LIN {X 0.261,Y -522.750,Z 821.053,A 0.000,B 0.000,C 90.000,E1 45.567} C_DIS
LIN {X -0.024,Y -519.538,Z 821.051,A 0.000,B 0.000,C 90.000,E1 45.162} C_DIS
LIN {X -0.181,Y -514.770,Z 821.048,A 0.000,B 0.000,C 90.000,E1 44.595} C_DIS
LIN {X -0.024,Y -506.960,Z 821.043,A 0.000,B 0.000,C 90.000,E1 43.704} C_DIS
LIN {X -0.047,Y -501.436,Z 821.040,A 0.000,B 0.000,C 90.000,E1 43.137} C_DIS
LIN {X 0.036,Y -494.169,Z 821.036,A 0.000,B 0.000,C 90.000,E1 42.447} C_DIS
LIN {X -0.150,Y -491.333,Z 821.034,A 0.000,B 0.000,C 90.000,E1 42.204} C_DIS
LIN {X 0.096,Y -483.937,Z 821.031,A 0.000,B 0.000,C 90.000,E1 41.553} C_DIS
LIN {X 0.088,Y -474.648,Z 821.027,A 0.000,B 0.000,C 90.000,E1 40.825} C_DIS
LIN {X -0.048,Y -466.706,Z 821.024,A 0.000,B 0.000,C 90.000,E1 40.253} C_DIS
LIN {X 0.197,Y -452.653,Z 821.018,A 0.000,B 0.000,C 90.000,E1 39.197} C_DIS
LIN {X -0.100,Y -425.883,Z 821.007,A 0.000,B 0.000,C 90.000,E1 37.237} C_DIS
LIN {X 0.137,Y -410.645,Z 821.000,A 0.000,B 0.000,C 90.000,E1 35.931} C_DIS
LIN {X -0.191,Y -403.603,Z 820.996,A 0.000,B 0.000,C 90.000,E1 35.311} C_DIS
LIN {X -0.106,Y -398.523,Z 820.993,A 0.000,B 0.000,C 90.000,E1 34.739} C_DIS
LIN {X -0.162,Y -398.192,Z 820.993,A 0.000,B 0.000,C 90.000,E1 34.692} C_DIS
LIN {X 0.030,Y -398.175,Z 820.993,A 0.000,B 0.000,C 90.000,E1 34.659} C_DIS
LIN {X -0.048,Y -393.629,Z 820.976,A 0.000,B 0.000,C 90.000,E1 31.750} C_DIS
LIN {X -0.048,Y -392.420,Z 820.973,A 0.000,B 0.000,C 90.000,E1 31.131} C_DIS
LIN {X -0.226,Y -393.696,Z 820.957,A 0.000,B 0.000,C 90.000,E1 28.231} C_DIS
LIN {X 0.009,Y -395.185,Z 820.943,A 0.000,B 0.000,C 90.000,E1 25.720} C_DIS
LIN {X -0.060,Y -396.928,Z 820.929,A 0.000,B 0.000,C 90.000,E1 23.259} C_DIS
LIN {X -0.026,Y -398.855,Z 820.916,A 0.000,B 0.000,C 90.000,E1 20.791} C_DIS
LIN {X 0.052,Y -402.408,Z 820.896,A 0.000,B 0.000,C 90.000,E1 17.275} C_DIS
LIN {X -0.086,Y -407.529,Z 820.875,A 0.000,B 0.000,C 90.000,E1 13.467} C_DIS
LIN {X 0.213,Y -411.448,Z 820.861,A 0.000,B 0.000,C 90.000,E1 11.007} C_DIS
LIN {X 0.068,Y -415.594,Z 820.848,A 0.000,B 0.000,C 90.000,E1 8.624} C_DIS
LIN {X -0.139,Y -419.301,Z 820.837,A 0.000,B 0.000,C 90.000,E1 6.606} C_DIS
LIN {X 0.165,Y -423.039,Z 820.825,A 0.000,B 0.000,C 90.000,E1 4.531} C_DIS
LIN {X 0.185,Y -428.270,Z 820.810,A 0.000,B 0.000,C 90.000,E1 1.835} C_DIS
LIN {X -0.100,Y -434.151,Z 820.795,A 0.000,B 0.000,C 90.000,E1 359.141} C_DIS
LIN {X -0.156,Y -440.322,Z 820.781,A 0.000,B 0.000,C 90.000,E1 356.502} C_DIS
LIN {X 0.201,Y -445.132,Z 820.770,A 0.000,B 0.000,C 90.000,E1 354.489} C_DIS
LIN {X -0.223,Y -450.092,Z 820.759,A 0.000,B 0.000,C 90.000,E1 352.591} C_DIS
LIN {X 0.120,Y -453.638,Z 820.752,A 0.000,B 0.000,C 90.000,E1 351.254} C_DIS
LIN {X -0.050,Y -455.247,Z 820.749,A 0.000,B 0.000,C 90.000,E1 350.792} C_DIS
LIN {X 0.167,Y -456.464,Z 820.747,A 0.000,B 0.000,C 90.000,E1 350.443} C_DIS
LIN {X 0.216,Y -458.621,Z 820.745,A 0.000,B 0.000,C 90.000,E1 350.038} C_DIS
LIN {X -0.035,Y -462.489,Z 820.742,A 0.000,B 0.000,C 90.000,E1 349.567} C_DIS
LIN {X -0.211,Y -468.707,Z 820.739,A 0.000,B 0.000,C 90.000,E1 349.050} C_DIS
LIN {X 0.158,Y -479.221,Z 820.735,A 0.000,B 0.000,C 90.000,E1 348.285} C_DIS
LIN {X 0.243,Y -491.872,Z 820.731,A 0.000,B 0.000,C 90.000,E1 347.465} C_DIS
LIN {X -0.043,Y -501.420,Z 820.727,A 0.000,B 0.000,C 90.000,E1 346.881} C_DIS
LIN {X 0.173,Y -512.520,Z 820.723,A 0.000,B 0.000,C 90.000,E1 346.117} C_DIS
LIN {X -0.111,Y -524.906,Z 820.718,A 0.000,B 0.000,C 90.000,E1 345.283} C_DIS
LIN {X -0.145,Y -535.618,Z 820.714,A 0.000,B 0.000,C 90.000,E1 344.519} C_DIS
LIN {X -0.182,Y -544.323,Z 820.710,A 0.000,B 0.000,C 90.000,E1 343.850} C_DIS
LIN {X -0.257,Y -551.470,Z 820.707,A 0.000,B 0.000,C 90.000,E1 343.268} C_DIS
LIN {X -0.288,Y -559.767,Z 820.703,A 0.000,B 0.000,C 90.000,E1 342.543} C_DIS
LIN {X 0.011,Y -566.278,Z 820.699,A 0.000,B 0.000,C 90.000,E1 341.873} C_DIS
LIN {X 0.207,Y -571.344,Z 820.696,A 0.000,B 0.000,C 90.000,E1 341.329} C_DIS
LIN {X -0.071,Y -577.480,Z 820.693,A 0.000,B 0.000,C 90.000,E1 340.678} C_DIS
LIN {X 0.221,Y -580.873,Z 820.690,A 0.000,B 0.000,C 90.000,E1 340.242} C_DIS
LIN {X 0.266,Y -585.084,Z 820.687,A 0.000,B 0.000,C 90.000,E1 339.699} C_DIS
LIN {X -0.213,Y -589.010,Z 820.684,A 0.000,B 0.000,C 90.000,E1 339.209} C_DIS
LIN {X 0.096,Y -592.676,Z 820.681,A 0.000,B 0.000,C 90.000,E1 338.646} C_DIS
LIN {X 0.217,Y -596.076,Z 820.679,A 0.000,B 0.000,C 90.000,E1 338.103} C_DIS
LIN {X 0.122,Y -604.108,Z 820.671,A 0.000,B 0.000,C 90.000,E1 336.794} C_DIS
LIN {X 0.182,Y -611.002,Z 820.665,A 0.000,B 0.000,C 90.000,E1 335.613} C_DIS
LIN {X 0.055,Y -616.881,Z 820.659,A 0.000,B 0.000,C 90.000,E1 334.588} C_DIS
LIN {X 0.011,Y -622.293,Z 820.653,A 0.000,B 0.000,C 90.000,E1 333.563} C_DIS
LIN {X 0.034,Y -626.798,Z 820.648,A 0.000,B 0.000,C 90.000,E1 332.666} C_DIS
LIN {X 0.117,Y -631.547,Z 820.643,A 0.000,B 0.000,C 90.000,E1 331.641} C_DIS
LIN {X -0.346,Y -635.033,Z 820.638,A 0.000,B 0.000,C 90.000,E1 330.923} C_DIS
LIN {X 0.191,Y -640.656,Z 820.631,A 0.000,B 0.000,C 90.000,E1 329.616} C_DIS
LIN {X 0.198,Y -644.703,Z 820.626,A 0.000,B 0.000,C 90.000,E1 328.614} C_DIS
LIN {X -0.292,Y -648.527,Z 820.620,A 0.000,B 0.000,C 90.000,E1 327.661} C_DIS
LIN {X -0.265,Y -651.215,Z 820.616,A 0.000,B 0.000,C 90.000,E1 326.914} C_DIS
LIN {X 0.229,Y -656.062,Z 820.608,A 0.000,B 0.000,C 90.000,E1 325.388} C_DIS
LIN {X -0.214,Y -658.277,Z 820.604,A 0.000,B 0.000,C 90.000,E1 324.689} C_DIS
LIN {X 0.284,Y -660.412,Z 820.600,A 0.000,B 0.000,C 90.000,E1 323.909} C_DIS
LIN {X -0.075,Y -663.725,Z 820.593,A 0.000,B 0.000,C 90.000,E1 322.718} C_DIS
LIN {X 0.008,Y -666.596,Z 820.586,A 0.000,B 0.000,C 90.000,E1 321.492} C_DIS
LIN {X 0.041,Y -669.225,Z 820.579,A 0.000,B 0.000,C 90.000,E1 320.275} C_DIS
LIN {X 0.123,Y -671.181,Z 820.574,A 0.000,B 0.000,C 90.000,E1 319.299} C_DIS
LIN {X -0.189,Y -673.898,Z 820.566,A 0.000,B 0.000,C 90.000,E1 317.877} C_DIS
LIN {X -0.149,Y -674.733,Z 820.563,A 0.000,B 0.000,C 90.000,E1 317.391} C_DIS
LIN {X -0.071,Y -675.827,Z 820.559,A 0.000,B 0.000,C 90.000,E1 316.662} C_DIS
LIN {X -0.412,Y -677.302,Z 820.554,A 0.000,B 0.000,C 90.000,E1 315.729} C_DIS
LIN {X -0.267,Y -678.550,Z 820.549,A 0.000,B 0.000,C 90.000,E1 314.757} C_DIS
LIN {X -0.065,Y -680.027,Z 820.542,A 0.000,B 0.000,C 90.000,E1 313.542} C_DIS
LIN {X 0.238,Y -681.705,Z 820.534,A 0.000,B 0.000,C 90.000,E1 312.081} C_DIS
LIN {X -0.386,Y -683.274,Z 820.526,A 0.000,B 0.000,C 90.000,E1 310.701} C_DIS
LIN {X -0.033,Y -684.739,Z 820.518,A 0.000,B 0.000,C 90.000,E1 309.241} C_DIS
LIN {X 0.011,Y -686.073,Z 820.510,A 0.000,B 0.000,C 90.000,E1 307.810} C_DIS
LIN {X 0.127,Y -687.483,Z 820.501,A 0.000,B 0.000,C 90.000,E1 306.137} C_DIS
LIN {X -0.176,Y -688.595,Z 820.493,A 0.000,B 0.000,C 90.000,E1 304.739} C_DIS
LIN {X 0.113,Y -689.593,Z 820.485,A 0.000,B 0.000,C 90.000,E1 303.293} C_DIS
LIN {X -0.310,Y -690.785,Z 820.476,A 0.000,B 0.000,C 90.000,E1 301.671} C_DIS
LIN {X -0.220,Y -691.520,Z 820.471,A 0.000,B 0.000,C 90.000,E1 300.718} C_DIS
LIN {X -0.364,Y -692.668,Z 820.461,A 0.000,B 0.000,C 90.000,E1 299.077} C_DIS
LIN {X -0.116,Y -693.655,Z 820.454,A 0.000,B 0.000,C 90.000,E1 297.641} C_DIS
LIN {X 0.082,Y -694.959,Z 820.444,A 0.000,B 0.000,C 90.000,E1 295.976} C_DIS
LIN {X -0.245,Y -696.093,Z 820.437,A 0.000,B 0.000,C 90.000,E1 294.591} C_DIS
LIN {X 0.010,Y -696.285,Z 820.435,A 0.000,B 0.000,C 90.000,E1 294.335} C_DIS
LIN {X -0.398,Y -696.241,Z 820.433,A 0.000,B 0.000,C 90.000,E1 293.898} C_DIS
LIN {X -0.143,Y -696.109,Z 820.431,A 0.000,B 0.000,C 90.000,E1 293.643} C_DIS
LIN {X 0.088,Y -695.005,Z 820.429,A 0.000,B 0.000,C 90.000,E1 293.153} C_DIS
LIN {X -0.301,Y -694.188,Z 820.427,A 0.000,B 0.000,C 90.000,E1 292.950} C_DIS
LIN {X -0.177,Y -693.397,Z 820.427,A 0.000,B 0.000,C 90.000,E1 292.823} C_DIS
LIN {X -0.201,Y -691.404,Z 820.425,A 0.000,B 0.000,C 90.000,E1 292.589} C_DIS
LIN {X 0.038,Y -689.032,Z 820.424,A 0.000,B 0.000,C 90.000,E1 292.333} C_DIS
LIN {X 0.155,Y -687.607,Z 820.423,A 0.000,B 0.000,C 90.000,E1 292.206} C_DIS
LIN {X -0.272,Y -683.409,Z 820.422,A 0.000,B 0.000,C 90.000,E1 292.025} C_DIS
LIN {X 0.129,Y -677.903,Z 820.421,A 0.000,B 0.000,C 90.000,E1 291.770} C_DIS
LIN {X 0.332,Y -672.231,Z 820.420,A 0.000,B 0.000,C 90.000,E1 291.589} C_DIS
LIN {X 0.142,Y -661.046,Z 820.419,A 0.000,B 0.000,C 90.000,E1 291.408} C_DIS
LIN {X 0.053,Y -645.225,Z 820.418,A 0.000,B 0.000,C 90.000,E1 291.153} C_DIS
LIN {X -0.171,Y -634.737,Z 820.417,A 0.000,B 0.000,C 90.000,E1 290.972} C_DIS
LIN {X -0.106,Y -625.306,Z 820.415,A 0.000,B 0.000,C 90.000,E1 290.737} C_DIS
LIN {X -0.279,Y -620.218,Z 820.414,A 0.000,B 0.000,C 90.000,E1 290.610} C_DIS
LIN {X -0.208,Y -615.713,Z 820.413,A 0.000,B 0.000,C 90.000,E1 290.429} C_DIS
LIN {X -0.183,Y -610.222,Z 820.412,A 0.000,B 0.000,C 90.000,E1 290.174} C_DIS
LIN {X -0.008,Y -607.280,Z 820.411,A 0.000,B 0.000,C 90.000,E1 289.939} C_DIS
LIN {X -0.044,Y -607.237,Z 820.411,A 0.000,B 0.000,C 90.000,E1 289.939} C_DIS
LIN {X -0.081,Y -606.527,Z 820.410,A 0.000,B 0.000,C 90.000,E1 289.812} C_DIS
LIN {X -0.117,Y -606.510,Z 820.410,A 0.000,B 0.000,C 90.000,E1 289.812} C_DIS
LIN {X 0.208,Y -607.485,Z 820.408,A 0.000,B 0.000,C 90.000,E1 289.322} C_DIS
LIN {X -0.028,Y -608.040,Z 820.407,A 0.000,B 0.000,C 90.000,E1 289.214} C_DIS
LIN {X -0.067,Y -612.803,Z 820.402,A 0.000,B 0.000,C 90.000,E1 288.417} C_DIS
LIN {X 0.205,Y -616.014,Z 820.399,A 0.000,B 0.000,C 90.000,E1 287.873} C_DIS
LIN {X -0.301,Y -619.279,Z 820.396,A 0.000,B 0.000,C 90.000,E1 287.275} C_DIS
LIN {X -0.212,Y -622.448,Z 820.392,A 0.000,B 0.000,C 90.000,E1 286.496} C_DIS
LIN {X -0.050,Y -624.272,Z 820.389,A 0.000,B 0.000,C 90.000,E1 285.969} C_DIS
LIN {X 0.090,Y -626.626,Z 820.384,A 0.000,B 0.000,C 90.000,E1 285.190} C_DIS
LIN {X 0.091,Y -628.257,Z 820.380,A 0.000,B 0.000,C 90.000,E1 284.426} C_DIS
LIN {X -0.151,Y -629.151,Z 820.377,A 0.000,B 0.000,C 90.000,E1 283.939} C_DIS
LIN {X 0.068,Y -629.657,Z 820.375,A 0.000,B 0.000,C 90.000,E1 283.411} C_DIS
LIN {X 0.098,Y -629.974,Z 820.370,A 0.000,B 0.000,C 90.000,E1 282.647} C_DIS
LIN {X 0.326,Y -629.753,Z 820.368,A 0.000,B 0.000,C 90.000,E1 282.119} C_DIS
LIN {X 0.230,Y -628.573,Z 820.363,A 0.000,B 0.000,C 90.000,E1 281.366} C_DIS
LIN {X -0.167,Y -627.488,Z 820.360,A 0.000,B 0.000,C 90.000,E1 280.894} C_DIS
LIN {X 0.043,Y -626.083,Z 820.358,A 0.000,B 0.000,C 90.000,E1 280.366} C_DIS
LIN {X 0.132,Y -624.391,Z 820.355,A 0.000,B 0.000,C 90.000,E1 279.849} C_DIS
LIN {X 0.154,Y -621.521,Z 820.351,A 0.000,B 0.000,C 90.000,E1 279.208} C_DIS
LIN {X 0.218,Y -618.801,Z 820.348,A 0.000,B 0.000,C 90.000,E1 278.690} C_DIS
LIN {X -0.256,Y -615.496,Z 820.346,A 0.000,B 0.000,C 90.000,E1 278.219} C_DIS
LIN {X -0.232,Y -611.361,Z 820.343,A 0.000,B 0.000,C 90.000,E1 277.701} C_DIS
LIN {X 0.112,Y -608.987,Z 820.341,A 0.000,B 0.000,C 90.000,E1 277.409} C_DIS
LIN {X -0.293,Y -605.067,Z 820.339,A 0.000,B 0.000,C 90.000,E1 277.068} C_DIS
LIN {X 0.169,Y -601.813,Z 820.338,A 0.000,B 0.000,C 90.000,E1 276.777} C_DIS
LIN {X -0.111,Y -597.017,Z 820.336,A 0.000,B 0.000,C 90.000,E1 276.486} C_DIS
LIN {X 0.278,Y -593.542,Z 820.335,A 0.000,B 0.000,C 90.000,E1 276.258} C_DIS
LIN {X -0.079,Y -586.727,Z 820.333,A 0.000,B 0.000,C 90.000,E1 275.967} C_DIS
LIN {X -0.101,Y -579.558,Z 820.332,A 0.000,B 0.000,C 90.000,E1 275.682} C_DIS
LIN {X -0.300,Y -574.108,Z 820.331,A 0.000,B 0.000,C 90.000,E1 275.511} C_DIS
LIN {X 0.241,Y -568.214,Z 820.330,A 0.000,B 0.000,C 90.000,E1 275.334} C_DIS
LIN {X -0.041,Y -565.945,Z 820.330,A 0.000,B 0.000,C 90.000,E1 275.334} C_DIS
LIN {X -0.144,Y -560.728,Z 820.330,A 0.000,B 0.000,C 90.000,E1 275.334} C_DIS
LIN {X -0.192,Y -552.749,Z 820.330,A 0.000,B 0.000,C 90.000,E1 275.334} C_DIS
LIN {X 0.154,Y -551.386,Z 820.329,A 0.000,B 0.000,C 90.000,E1 275.277} C_DIS
LIN {X 0.103,Y -551.194,Z 820.329,A 0.000,B 0.000,C 90.000,E1 275.277} C_DIS
LIN {X -0.190,Y -550.374,Z 820.328,A 0.000,B 0.000,C 90.000,E1 274.992} C_DIS
LIN {X 0.108,Y -549.844,Z 820.327,A 0.000,B 0.000,C 90.000,E1 274.821} C_DIS
LIN {X 0.131,Y -548.673,Z 820.320,A 0.000,B 0.000,C 90.000,E1 273.555} C_DIS
LIN {X -0.197,Y -547.941,Z 820.314,A 0.000,B 0.000,C 90.000,E1 272.465} C_DIS
LIN {X 0.140,Y -546.544,Z 820.303,A 0.000,B 0.000,C 90.000,E1 270.458} C_DIS
LIN {X -0.116,Y -545.149,Z 820.292,A 0.000,B 0.000,C 90.000,E1 268.511} C_DIS
LIN {X 0.198,Y -543.617,Z 820.279,A 0.000,B 0.000,C 90.000,E1 266.216} C_DIS
LIN {X -0.162,Y -542.916,Z 820.273,A 0.000,B 0.000,C 90.000,E1 265.122} C_DIS
LIN {X 0.016,Y -542.212,Z 820.267,A 0.000,B 0.000,C 90.000,E1 263.970} C_DIS
LIN {X 0.183,Y -541.023,Z 820.259,A 0.000,B 0.000,C 90.000,E1 262.534} C_DIS
LIN {X 0.070,Y -539.240,Z 820.248,A 0.000,B 0.000,C 90.000,E1 260.557} C_DIS
LIN {X -0.209,Y -537.837,Z 820.240,A 0.000,B 0.000,C 90.000,E1 259.162} C_DIS
LIN {X 0.172,Y -536.111,Z 820.230,A 0.000,B 0.000,C 90.000,E1 257.409} C_DIS
LIN {X 0.000,Y -534.946,Z 820.224,A 0.000,B 0.000,C 90.000,E1 256.284} C_DIS
LIN {X -0.091,Y -533.009,Z 820.214,A 0.000,B 0.000,C 90.000,E1 254.574} C_DIS
LIN {X 0.059,Y -531.046,Z 820.205,A 0.000,B 0.000,C 90.000,E1 252.834} C_DIS
LIN {X -0.030,Y -529.620,Z 820.198,A 0.000,B 0.000,C 90.000,E1 251.692} C_DIS
LIN {X 0.034,Y -527.818,Z 820.190,A 0.000,B 0.000,C 90.000,E1 250.242} C_DIS
LIN {X 0.239,Y -525.825,Z 820.182,A 0.000,B 0.000,C 90.000,E1 248.773} C_DIS
LIN {X 0.078,Y -523.323,Z 820.173,A 0.000,B 0.000,C 90.000,E1 247.050} C_DIS
LIN {X 0.054,Y -520.640,Z 820.163,A 0.000,B 0.000,C 90.000,E1 245.305} C_DIS
LIN {X 0.046,Y -518.257,Z 820.155,A 0.000,B 0.000,C 90.000,E1 243.845} C_DIS
LIN {X 0.225,Y -515.807,Z 820.147,A 0.000,B 0.000,C 90.000,E1 242.359} C_DIS
LIN {X 0.258,Y -512.535,Z 820.137,A 0.000,B 0.000,C 90.000,E1 240.589} C_DIS
LIN {X -0.223,Y -509.295,Z 820.127,A 0.000,B 0.000,C 90.000,E1 238.869} C_DIS
LIN {X -0.033,Y -506.926,Z 820.120,A 0.000,B 0.000,C 90.000,E1 237.661} C_DIS
LIN {X 0.079,Y -505.097,Z 820.115,A 0.000,B 0.000,C 90.000,E1 236.755} C_DIS
LIN {X 0.079,Y -501.835,Z 820.107,A 0.000,B 0.000,C 90.000,E1 235.261} C_DIS
LIN {X -0.115,Y -498.367,Z 820.099,A 0.000,B 0.000,C 90.000,E1 233.783} C_DIS
LIN {X 0.194,Y -496.211,Z 820.094,A 0.000,B 0.000,C 90.000,E1 232.844} C_DIS
LIN {X 0.042,Y -491.807,Z 820.084,A 0.000,B 0.000,C 90.000,E1 231.045} C_DIS
LIN {X 0.010,Y -486.114,Z 820.070,A 0.000,B 0.000,C 90.000,E1 228.609} C_DIS
LIN {X 0.008,Y -481.209,Z 820.058,A 0.000,B 0.000,C 90.000,E1 226.458} C_DIS
LIN {X -0.164,Y -478.457,Z 820.051,A 0.000,B 0.000,C 90.000,E1 225.243} C_DIS
LIN {X 0.299,Y -475.791,Z 820.044,A 0.000,B 0.000,C 90.000,E1 223.947} C_DIS
LIN {X -0.187,Y -472.437,Z 820.036,A 0.000,B 0.000,C 90.000,E1 222.447} C_DIS
LIN {X 0.044,Y -468.487,Z 820.025,A 0.000,B 0.000,C 90.000,E1 220.539} C_DIS
